	{attribute 'TcIecLibraryType'}
	{attribute 'external_name' := 'F_VN_Homography_GUID_BACE21C2_AF59_42BD_5B50_39109165FCFC'}
	(* Find the homography (perspective transformation) between two planar point sets. *)
	FUNCTION F_VN_Homography : HRESULT
	VAR_INPUT
		ipSrcPoints	:	ITcVnContainer;	(* Container with at least 4 source points (ContainerType_Vector_TcVnPoint2_REAL) *)
		ipDestPoints	:	ITcVnContainer;	(* Container with destination points (same number as ipSrcPoints, ContainerType_Vector_TcVnPoint2_REAL) *)
		aPerspectiveTransform	:	REFERENCE TO TcVnMatrix3x3_LREAL;	(* Returns the perspective transformation matrix, which transforms the source points to the destination points *)
		hrPrev	:	HRESULT;	(* HRESULT indicating the result of previous operations (If SUCCEEDED(hrPrev) equals false, no operation is executed.) *)
	END_VAR

END_FUNCTION

// Functions/Geometric and Coordinate Transformations/F_VN_HomographyExp

	{attribute 'TcIecLibraryType'}
	{attribute 'external_name' := 'F_VN_HomographyExp_GUID_957B3768_7821_437F_6422_7D349715F2AB'}
	(* Find the homography (perspective transformation) between two planar point sets. (expert function) *)
	FUNCTION F_VN_HomographyExp : HRESULT
	VAR_INPUT
		ipSrcPoints	:	ITcVnContainer;	(* Container with at least 4 source points (ContainerType_Vector_TcVnPoint2_REAL) *)
		ipDestPoints	:	ITcVnContainer;	(* Container with destination points (same number as ipSrcPoints, ContainerType_Vector_TcVnPoint2_REAL) *)
		aPerspectiveTransform	:	REFERENCE TO TcVnMatrix3x3_LREAL;	(* Returns the perspective transformation matrix, which transforms the source points to the destination points *)
		eAlgorithm	:	ETcVnEstimationAlgorithm;	(* Estimation algorithm *)
		fReprojThreshold	:	LREAL;	(* Maximum allowed reprojection error to treat a point pair as an inlier (only for RANSAC, RHO) *)
		ipInlierMask	:	REFERENCE TO ITcVnContainer;	(* Returns a mask marking the inliers (optional, set to 0 if not required; ContainerType_Vector_SINT; only for RANSAC, LMEDS) *)
		nMaxIterations	:	UDINT;	(* Maximum number of RANSAC iterations *)
		fConfidence	:	LREAL;	(* Confidence (0..1) *)
		hrPrev	:	HRESULT;	(* HRESULT indicating the result of previous operations (If SUCCEEDED(hrPrev) equals false, no operation is executed.) *)
	END_VAR

END_FUNCTION

// Functions/Geometric and Coordinate Transformations/F_VN_ImagePointsWorldDistance

	{attribute 'TcIecLibraryType'}
	{attribute 'external_name' := 'F_VN_ImagePointsWorldDistance_GUID_B7CC4CD8_D9B9_453D_47E9_DCE0997F3FF0'}
	(* Computes the distance in the world coordinate system between two points (in the same world coordinate z layer) given in image coordinates. *)
	FUNCTION F_VN_ImagePointsWorldDistance : HRESULT
	VAR_INPUT
		aImagePoint1	:	REFERENCE TO TcVnPoint2_REAL;	(* First point in the image coordinate system *)
		aImagePoint2	:	REFERENCE TO TcVnPoint2_REAL;	(* Second point in the image coordinate system *)
		fWorldDistance	:	REFERENCE TO LREAL;	(* Returns the distance between aImagePoint1 and aImagePoint2 in the world coordinate system *)
		aCameraMatrix	:	REFERENCE TO TcVnMatrix3x3_LREAL;	(* 3x3 camera matrix containing the intrinsic parameters *)
		aDistortionCoefficients	:	REFERENCE TO TcVnArray8_LREAL;	(* Lens distortion coefficients [k1, k2, p1, p2, k3, k4, k5, k6] *)
		aRotationMatrix	:	REFERENCE TO TcVnMatrix3x3_LREAL;	(* 3x3 rotation matrix *)
		aTranslationVector	:	REFERENCE TO TcVnVector3_LREAL;	(* Translation vector *)
		fZ	:	LREAL;	(* z coordinate (world coordinate system) of the given points (0 would be at (toplevel) calibration pattern) *)
		hrPrev	:	HRESULT;	(* HRESULT indicating the result of previous operations (If SUCCEEDED(hrPrev) equals false, no operation is executed.) *)
	END_VAR

END_FUNCTION

// Functions/Geometric and Coordinate Transformations/F_VN_InvertAffineTransformation

	{attribute 'TcIecLibraryType'}
	{attribute 'external_name' := 'F_VN_InvertAffineTransformation_GUID_9CD3C3CD_AED1_4AC7_6B76_3AB059F5DF24'}
	(* Invert a 2D affine transformation matrix. *)
	FUNCTION F_VN_InvertAffineTransformation : HRESULT
	VAR_INPUT
		aTransformationMatrix	:	REFERENCE TO TcVnMatrix2x3_LREAL;	(* Source affine transformation matrix *)
		aInvertedTransformationMatrix	:	REFERENCE TO TcVnMatrix2x3_LREAL;	(* Resulting inverted affine transformation matrix *)
		hrPrev	:	HRESULT;	(* HRESULT indicating the result of previous operations (If SUCCEEDED(hrPrev) equals false, no operation is executed.) *)
	END_VAR

END_FUNCTION

// Functions/Geometric and Coordinate Transformations/F_VN_PerspectiveTransformation

	{attribute 'TcIecLibraryType'}
	{attribute 'external_name' := 'F_VN_PerspectiveTransformation_GUID_A10BDBDF_3A4E_42F2_67E8_D12DFF09F118'}
	(* Apply a perspective transformation (rotation + translation, e.g. from extrinsic calibration) to 3D point coordinates. *)
	FUNCTION F_VN_PerspectiveTransformation : HRESULT
	VAR_INPUT
		ipSrcPoints	:	ITcVnContainer;	(* Container with 3D source points (TcVnPoint3_REAL or TcVnPoint3_LREAL) *)
		ipDestPoints	:	REFERENCE TO ITcVnContainer;	(* Returns the transformed points (same type as ipSrcPoints) *)
		aRotationMatrix	:	REFERENCE TO TcVnMatrix3x3_LREAL;	(* 3x3 rotation matrix *)
		aTranslationVector	:	REFERENCE TO TcVnVector3_LREAL;	(* Translation vector *)
		hrPrev	:	HRESULT;	(* HRESULT indicating the result of previous operations (If SUCCEEDED(hrPrev) equals false, no operation is executed.) *)
	END_VAR

END_FUNCTION

// Functions/Geometric and Coordinate Transformations/F_VN_PyramidDown

	{attribute 'TcIecLibraryType'}
	{attribute 'external_name' := 'F_VN_PyramidDown_GUID_A46C393D_F610_403D_7A8C_F077AAEC78D7'}
	(* Downsamples an image to half width and height. *)
	FUNCTION F_VN_PyramidDown : HRESULT
	VAR_INPUT
		ipSrcImage	:	ITcVnImage;	(* Source image *)
		ipDestImage	:	REFERENCE TO ITcVnImage;	(* Destination image (An appropriate destination image will be created if required.) *)
		hrPrev	:	HRESULT;	(* HRESULT indicating the result of previous operations (If SUCCEEDED(hrPrev) equals false, no operation is executed.) *)
	END_VAR

END_FUNCTION

// Functions/Geometric and Coordinate Transformations/F_VN_PyramidUp

	{attribute 'TcIecLibraryType'}
	{attribute 'external_name' := 'F_VN_PyramidUp_GUID_C7623CD4_6E7C_4659_6255_40F31BC5DBAD'}
	(* Upsamples an image to double width and height. *)
	FUNCTION F_VN_PyramidUp : HRESULT
	VAR_INPUT
		ipSrcImage	:	ITcVnImage;	(* Source image *)
		ipDestImage	:	REFERENCE TO ITcVnImage;	(* Destination image (An appropriate destination image will be created if required.) *)
		hrPrev	:	HRESULT;	(* HRESULT indicating the result of previous operations (If SUCCEEDED(hrPrev) equals false, no operation is executed.) *)
	END_VAR

END_FUNCTION

// Functions/Geometric and Coordinate Transformations/F_VN_RemapImageToLogPolarSpace

	{attribute 'TcIecLibraryType'}
	{attribute 'external_name' := 'F_VN_RemapImageToLogPolarSpace_GUID_317EBF55_4B2D_478D_5790_D67FEE90C80E'}
	(* Remap an image to log-polar space. *)
	FUNCTION F_VN_RemapImageToLogPolarSpace : HRESULT
	VAR_INPUT
		ipSrcImage	:	ITcVnImage;	(* Source image *)
		ipDestImage	:	REFERENCE TO ITcVnImage;	(* Destination image (Must not be the same as ipSrcImage! An appropriate destination image will be created if required.) *)
		aCenter	:	REFERENCE TO TcVnPoint2_REAL;	(* Center point for the transformation *)
		hrPrev	:	HRESULT;	(* HRESULT indicating the result of previous operations (If SUCCEEDED(hrPrev) equals false, no operation is executed.) *)
	END_VAR

END_FUNCTION

// Functions/Geometric and Coordinate Transformations/F_VN_RemapImageToLogPolarSpaceExp

	{attribute 'TcIecLibraryType'}
	{attribute 'external_name' := 'F_VN_RemapImageToLogPolarSpaceExp_GUID_C452CB02_0761_45C6_6145_95B8240BC99B'}
	(* Remap an image to log-polar space. (expert function) *)
	FUNCTION F_VN_RemapImageToLogPolarSpaceExp : HRESULT
	VAR_INPUT
		ipSrcImage	:	ITcVnImage;	(* Source image *)
		ipDestImage	:	REFERENCE TO ITcVnImage;	(* Destination image (Must not be the same as ipSrcImage! An appropriate destination image will be created if required.) *)
		aCenter	:	REFERENCE TO TcVnPoint2_REAL;	(* Center point for the transformation *)
		fScale	:	LREAL;	(* Magnitude scale parameter (set to 0 for auto select) *)
		eInterpolationType	:	ETcVnInterpolationType;	(* Interpolation type *)
		hrPrev	:	HRESULT;	(* HRESULT indicating the result of previous operations (If SUCCEEDED(hrPrev) equals false, no operation is executed.) *)
	END_VAR

END_FUNCTION

// Functions/Geometric and Coordinate Transformations/F_VN_RemapImageToPolarSpace

	{attribute 'TcIecLibraryType'}
	{attribute 'external_name' := 'F_VN_RemapImageToPolarSpace_GUID_81A2C6C8_42C0_4CD4_568D_C8E6F1DB1310'}
	(* Remap an image to polar space. *)
	FUNCTION F_VN_RemapImageToPolarSpace : HRESULT
	VAR_INPUT
		ipSrcImage	:	ITcVnImage;	(* Source image *)
		ipDestImage	:	REFERENCE TO ITcVnImage;	(* Destination image (Must not be the same as ipSrcImage! An appropriate destination image will be created if required.) *)
		aCenter	:	REFERENCE TO TcVnPoint2_REAL;	(* Center point for the transformation *)
		hrPrev	:	HRESULT;	(* HRESULT indicating the result of previous operations (If SUCCEEDED(hrPrev) equals false, no operation is executed.) *)
	END_VAR

END_FUNCTION

// Functions/Geometric and Coordinate Transformations/F_VN_RemapImageToPolarSpaceExp

	{attribute 'TcIecLibraryType'}
	{attribute 'external_name' := 'F_VN_RemapImageToPolarSpaceExp_GUID_C787DB85_1BF7_45E0_4B56_DABB0704543F'}
	(* Remap an image to polar space. (expert function) *)
	FUNCTION F_VN_RemapImageToPolarSpaceExp : HRESULT
	VAR_INPUT
		ipSrcImage	:	ITcVnImage;	(* Source image *)
		ipDestImage	:	REFERENCE TO ITcVnImage;	(* Destination image (Must not be the same as ipSrcImage! An appropriate destination image will be created if required.) *)
		aCenter	:	REFERENCE TO TcVnPoint2_REAL;	(* Center point for the transformation *)
		fMaxRadius	:	LREAL;	(* Maximum radius for the transformation (set to 0 for auto select) *)
		eInterpolationType	:	ETcVnInterpolationType;	(* Interpolation type *)
		hrPrev	:	HRESULT;	(* HRESULT indicating the result of previous operations (If SUCCEEDED(hrPrev) equals false, no operation is executed.) *)
	END_VAR

END_FUNCTION

// Functions/Geometric and Coordinate Transformations/F_VN_ResizeImage

	{attribute 'TcIecLibraryType'}
	{attribute 'external_name' := 'F_VN_ResizeImage_GUID_B297F5D8_147F_492A_69A8_8AF713B422F2'}
	(* Resize an image using a specific interpolation type. *)
	FUNCTION F_VN_ResizeImage : HRESULT
	VAR_INPUT
		ipSrcImage	:	ITcVnImage;	(* Source image *)
		ipDestImage	:	REFERENCE TO ITcVnImage;	(* Destination image (An appropriate image will be created if required.) *)
		nWidth	:	UDINT;	(* New width *)
		nHeight	:	UDINT;	(* New height *)
		eInterpolationType	:	ETcVnInterpolationType;	(* Interpolation type *)
		hrPrev	:	HRESULT;	(* HRESULT indicating the result of previous operations (If SUCCEEDED(hrPrev) equals false, no operation is executed.) *)
	END_VAR

END_FUNCTION

// Functions/Geometric and Coordinate Transformations/F_VN_RotateImage

	{attribute 'TcIecLibraryType'}
	{attribute 'external_name' := 'F_VN_RotateImage_GUID_D34C046F_1F65_490B_4694_D44E5095070F'}
	(* Rotate an image by 90, 180, or 270 degrees in clockwise direction. *)
	FUNCTION F_VN_RotateImage : HRESULT
	VAR_INPUT
		ipSrcImage	:	ITcVnImage;	(* Source image *)
		ipDestImage	:	REFERENCE TO ITcVnImage;	(* Destination image (An appropriate image will be created if required.) *)
		eAngle	:	ETcVnRotationAngle;	(* Rotation angle *)
		hrPrev	:	HRESULT;	(* HRESULT indicating the result of previous operations (If SUCCEEDED(hrPrev) equals false, no operation is executed.) *)
	END_VAR

END_FUNCTION

// Functions/Geometric and Coordinate Transformations/F_VN_WarpAffine

	{attribute 'TcIecLibraryType'}
	{attribute 'external_name' := 'F_VN_WarpAffine_GUID_2706E1B0_49AA_4EA6_4BCD_DBE188F95A14'}
	(* Apply an affine transformation to an image. *)
	FUNCTION F_VN_WarpAffine : HRESULT
	VAR_INPUT
		ipSrcImage	:	ITcVnImage;	(* Source image *)
		ipDestImage	:	REFERENCE TO ITcVnImage;	(* Destination image (An appropriate image will be created if required.) *)
		aTransformationMatrix	:	REFERENCE TO TcVnMatrix2x3_LREAL;	(* Affine transformation matrix *)
		hrPrev	:	HRESULT;	(* HRESULT indicating the result of previous operations (If SUCCEEDED(hrPrev) equals false, no operation is executed.) *)
	END_VAR

END_FUNCTION

// Functions/Geometric and Coordinate Transformations/F_VN_WarpAffineExp

	{attribute 'TcIecLibraryType'}
	{attribute 'external_name' := 'F_VN_WarpAffineExp_GUID_BA2CF855_8F8F_4276_5F6B_1E3D858121C1'}
	(* Apply an affine transformation to an image. (expert function) *)
	FUNCTION F_VN_WarpAffineExp : HRESULT
	VAR_INPUT
		ipSrcImage	:	ITcVnImage;	(* Source image *)
		ipDestImage	:	REFERENCE TO ITcVnImage;	(* Destination image (An appropriate image will be created if required.) *)
		aTransformationMatrix	:	REFERENCE TO TcVnMatrix2x3_LREAL;	(* Affine transformation matrix *)
		nDestWidth	:	UDINT;	(* Width of the destination image *)
		nDestHeight	:	UDINT;	(* Height of the destination image *)
		eInterpolationType	:	ETcVnInterpolationType;	(* Interpolation method *)
		bWarpInverse	:	BOOL;	(* Handle aTransformationMatrix as the inverse transformation *)
		eBorderInterpolation	:	ETcVnBorderInterpolationMethod;	(* Border interpolation method (ISOLATED not supported) *)
		fBorderValue	:	LREAL;	(* Border value, if CONSTANT is used *)
		hrPrev	:	HRESULT;	(* HRESULT indicating the result of previous operations (If SUCCEEDED(hrPrev) equals false, no operation is executed.) *)
	END_VAR

END_FUNCTION

// Functions/Geometric and Coordinate Transformations/F_VN_WarpAffine_Container

	{attribute 'TcIecLibraryType'}
	{attribute 'external_name' := 'F_VN_WarpAffine_Container_GUID_E245EF6B_F4F8_40CB_6A97_91315828A7CE'}
	(* Apply an affine transformation to a container of 2D points. *)
	FUNCTION F_VN_WarpAffine_Container : HRESULT
	VAR_INPUT
		ipSrcPoints	:	ITcVnContainer;	(* Source points (ContainerType_Vector_TcVnPoint2_DINT or ContainerType_Vector_TcVnPoint2_REAL or ContainerType_Vector_TcVnPoint2_LREAL) *)
		ipDestPoints	:	REFERENCE TO ITcVnContainer;	(* Returns the transformed points (same type ID as ipSrcPoints; Non-zero interface pointers are reused.) *)
		aTransformationMatrix	:	REFERENCE TO TcVnMatrix2x3_LREAL;	(* Affine transformation matrix *)
		hrPrev	:	HRESULT;	(* HRESULT indicating the result of previous operations (If SUCCEEDED(hrPrev) equals false, no operation is executed.) *)
	END_VAR

END_FUNCTION

// Functions/Geometric and Coordinate Transformations/F_VN_WarpAffine_Point

	{attribute 'TcIecLibraryType'}
	{attribute 'external_name' := 'F_VN_WarpAffine_Point_GUID_5382904B_C8E3_45B3_56E2_503ADF42779C'}
	(* Apply an affine transformation to a 2D point. *)
	FUNCTION F_VN_WarpAffine_Point : HRESULT
	VAR_INPUT
		aSrcPoint	:	REFERENCE TO TcVnPoint2_LREAL;	(* Source point *)
		aDestPoint	:	REFERENCE TO TcVnPoint2_LREAL;	(* Destination point *)
		aTransformationMatrix	:	REFERENCE TO TcVnMatrix2x3_LREAL;	(* Affine transformation matrix *)
		hrPrev	:	HRESULT;	(* HRESULT indicating the result of previous operations (If SUCCEEDED(hrPrev) equals false, no operation is executed.) *)
	END_VAR

END_FUNCTION

// Functions/Geometric and Coordinate Transformations/F_VN_WarpPerspective

	{attribute 'TcIecLibraryType'}
	{attribute 'external_name' := 'F_VN_WarpPerspective_GUID_A5B0ACEA_FF20_43BC_4699_A7DC79225D3D'}
	(* Apply a perspective transformation to an image. *)
	FUNCTION F_VN_WarpPerspective : HRESULT
	VAR_INPUT
		ipSrcImage	:	ITcVnImage;	(* Source image *)
		ipDestImage	:	REFERENCE TO ITcVnImage;	(* Destination image (An appropriate image will be created if required.) *)
		aTransformationMatrix	:	REFERENCE TO TcVnMatrix3x3_LREAL;	(* Perspective transformation matrix *)
		hrPrev	:	HRESULT;	(* HRESULT indicating the result of previous operations (If SUCCEEDED(hrPrev) equals false, no operation is executed.) *)
	END_VAR

END_FUNCTION

// Functions/Geometric and Coordinate Transformations/F_VN_WarpPerspectiveExp

	{attribute 'TcIecLibraryType'}
	{attribute 'external_name' := 'F_VN_WarpPerspectiveExp_GUID_5EE68E40_2F06_46A9_53D0_6833136D40D3'}
	(* Apply a perspective transformation to an image. (expert function) *)
	FUNCTION F_VN_WarpPerspectiveExp : HRESULT
	VAR_INPUT
		ipSrcImage	:	ITcVnImage;	(* Source image *)
		ipDestImage	:	REFERENCE TO ITcVnImage;	(* Destination image (An appropriate image will be created if required.) *)
		aTransformationMatrix	:	REFERENCE TO TcVnMatrix3x3_LREAL;	(* Perspective transformation matrix *)
		nDestWidth	:	UDINT;	(* Width of the destination image *)
		nDestHeight	:	UDINT;	(* Height of the destination image *)
		eInterpolationType	:	ETcVnInterpolationType;	(* Interpolation method *)
		bWarpInverse	:	BOOL;	(* Handle aTransformationMatrix as the inverse transformation *)
		eBorderInterpolation	:	ETcVnBorderInterpolationMethod;	(* Border interpolation method (ISOLATED not supported) *)
		fBorderValue	:	LREAL;	(* Border value, if CONSTANT is used *)
		hrPrev	:	HRESULT;	(* HRESULT indicating the result of previous operations (If SUCCEEDED(hrPrev) equals false, no operation is executed.) *)
	END_VAR

END_FUNCTION

// Functions/Geometric and Coordinate Transformations/F_VN_WarpPerspective_Point

	{attribute 'TcIecLibraryType'}
	{attribute 'external_name' := 'F_VN_WarpPerspective_Point_GUID_5538B106_075B_440A_4CE3_92BE11A2EC15'}
	(* Apply a perspective transformation to a 2D point. *)
	FUNCTION F_VN_WarpPerspective_Point : HRESULT
	VAR_INPUT
		aSrcPoint	:	REFERENCE TO TcVnPoint2_LREAL;	(* Source point *)
		aDestPoint	:	REFERENCE TO TcVnPoint2_LREAL;	(* Destination point *)
		aTransformationMatrix	:	REFERENCE TO TcVnMatrix3x3_LREAL;	(* Perspective transformation matrix *)
		hrPrev	:	HRESULT;	(* HRESULT indicating the result of previous operations (If SUCCEEDED(hrPrev) equals false, no operation is executed.) *)
	END_VAR

END_FUNCTION

// Functions/Contour Analysis/F_VN_ApproximatePolygon

	{attribute 'TcIecLibraryType'}
	{attribute 'external_name' := 'F_VN_ApproximatePolygon_GUID_CC2021C4_5F20_4D4F_750B_DA13A9B816C9'}
	(* Approximate a contour to a simplified polygon (using the Douglas-Peucker algorithm). *)
	FUNCTION F_VN_ApproximatePolygon : HRESULT
	VAR_INPUT
		ipSrcContour	:	ITcVnContainer;	(* Single contour (ContainerType_Vector_TcVnPoint2_DINT or ContainerType_Vector_TcVnPoint2_REAL; The elements of this container are the points of the contour.) *)
		ipDestContour	:	REFERENCE TO ITcVnContainer;	(* Returns a container which is filled with the approximated polygon points (same type ID as ipSrcContour; Non-zero interface pointers are reused.) *)
		fMaxDist	:	LREAL;	(* Maximum distance between the original contour and its approximation *)
		bClosed	:	BOOL;	(* Specify, if the contour is closed (first and last points connected) or not *)
		hrPrev	:	HRESULT;	(* HRESULT indicating the result of previous operations (If SUCCEEDED(hrPrev) equals false, no operation is executed.) *)
	END_VAR

END_FUNCTION

// Functions/Contour Analysis/F_VN_CheckIfPointIsInsideContour

	{attribute 'TcIecLibraryType'}
	{attribute 'external_name' := 'F_VN_CheckIfPointIsInsideContour_GUID_0925219F_5855_4324_6916_36F829EC1C7B'}
	(* Checks if a point is inside a contour (and optionally return the distance to it). *)
	FUNCTION F_VN_CheckIfPointIsInsideContour : HRESULT
	VAR_INPUT
		ipContour	:	ITcVnContainer;	(* Single contour (ContainerType_Vector_TcVnPoint2_DINT or ContainerType_Vector_TcVnPoint2_REAL) *)
		aPoint	:	REFERENCE TO TcVnPoint2_REAL;	(* Point position to check *)
		fDist	:	REFERENCE TO LREAL;	(* Returns the result (> 0: the point is inside the contour; 0: the point is on the contour; < 0: the point is outside the contour) *)
		bMeasureDistance	:	BOOL;	(* If true, fDist returns the distance to the nearest contour edge. Otherwise, fDist only returns -1, 0 or +1 (recommended to set to false if the distance is not required, as this is faster). *)
		hrPrev	:	HRESULT;	(* HRESULT indicating the result of previous operations (If SUCCEEDED(hrPrev) equals false, no operation is executed.) *)
	END_VAR

END_FUNCTION

// Functions/Contour Analysis/F_VN_ContourArea

	{attribute 'TcIecLibraryType'}
	{attribute 'external_name' := 'F_VN_ContourArea_GUID_D8EF7B56_DDD8_4A2A_43D3_6C64F8AEA3E5'}
	(* Estimate the contour area using Green's formula. *)
	FUNCTION F_VN_ContourArea : HRESULT
	VAR_INPUT
		ipContour	:	ITcVnContainer;	(* Single contour (ContainerType_Vector_TcVnPoint2_DINT or ContainerType_Vector_TcVnPoint2_REAL; The elements of this container are the points of the contour.) *)
		fArea	:	REFERENCE TO LREAL;	(* Returns the estimated contour area (The actual contour area may differ depending on the shape of the contour.) *)
		hrPrev	:	HRESULT;	(* HRESULT indicating the result of previous operations (If SUCCEEDED(hrPrev) equals false, no operation is executed.) *)
	END_VAR

END_FUNCTION

// Functions/Contour Analysis/F_VN_ContourCenterOfMass

	{attribute 'TcIecLibraryType'}
	{attribute 'external_name' := 'F_VN_ContourCenterOfMass_GUID_648B2107_798D_4ED5_549A_9A87656EE4D8'}
	(* Computes the center of mass of a contour. *)
	FUNCTION F_VN_ContourCenterOfMass : HRESULT
	VAR_INPUT
		ipContour	:	ITcVnContainer;	(* Single contour (ContainerType_Vector_TcVnPoint2_DINT or ContainerType_Vector_TcVnPoint2_REAL; The elements of this container are the points of the contour.) *)
		aCenterOfMass	:	REFERENCE TO TcVnPoint2_LREAL;	(* Returns the center of mass of the contour *)
		hrPrev	:	HRESULT;	(* HRESULT indicating the result of previous operations (If SUCCEEDED(hrPrev) equals false, no operation is executed.) *)
	END_VAR

END_FUNCTION

// Functions/Contour Analysis/F_VN_ContourCircularity

	{attribute 'TcIecLibraryType'}
	{attribute 'external_name' := 'F_VN_ContourCircularity_GUID_9E609700_7C0A_461F_5A42_99C7290586FE'}
	(* Computes the circularity of a contour (1.0: ideal circle, 0.0: straight line). *)
	FUNCTION F_VN_ContourCircularity : HRESULT
	VAR_INPUT
		ipContour	:	ITcVnContainer;	(* Single contour (ContainerType_Vector_TcVnPoint2_DINT or ContainerType_Vector_TcVnPoint2_REAL; The elements of this container are the points of the contour.) *)
		fCircularity	:	REFERENCE TO LREAL;	(* Returns the circularity of the contour [0..1] *)
		hrPrev	:	HRESULT;	(* HRESULT indicating the result of previous operations (If SUCCEEDED(hrPrev) equals false, no operation is executed.) *)
	END_VAR

END_FUNCTION

// Functions/Contour Analysis/F_VN_ContourEccentricity

	{attribute 'TcIecLibraryType'}
	{attribute 'external_name' := 'F_VN_ContourEccentricity_GUID_FFD20AEF_8984_4F5E_766E_3023FBFF4334'}
	(* Computes the eccentricity of a contour (0.0: circular, 1.0: linear). *)
	FUNCTION F_VN_ContourEccentricity : HRESULT
	VAR_INPUT
		ipContour	:	ITcVnContainer;	(* Single contour (ContainerType_Vector_TcVnPoint2_DINT or ContainerType_Vector_TcVnPoint2_REAL; The elements of this container are the points of the contour.) *)
		fEccentricity	:	REFERENCE TO LREAL;	(* Returns the eccentricity of the contour [0..1] *)
		hrPrev	:	HRESULT;	(* HRESULT indicating the result of previous operations (If SUCCEEDED(hrPrev) equals false, no operation is executed.) *)
	END_VAR

END_FUNCTION

// Functions/Contour Analysis/F_VN_ContourExtremePoint

	{attribute 'TcIecLibraryType'}
	{attribute 'external_name' := 'F_VN_ContourExtremePoint_GUID_8F761823_6FFC_4019_7B5F_2B40F751511F'}
	(* Finds the contour extreme point. *)
	FUNCTION F_VN_ContourExtremePoint : HRESULT
	VAR_INPUT
		ipContour	:	ITcVnContainer;	(* Source container with 2D points (TcVnPoint2_DINT or TcVnPoint2_REAL or TcVnPoint2_LREAL) *)
		eDirection	:	ETcVnExtremePointDirection;	(* Selects the search direction for the extreme point *)
		aExtremePoint	:	REFERENCE TO TcVnPoint2_LREAL;	(* Returns the extreme point of the contour, according to eDirection *)
		hrPrev	:	HRESULT;	(* HRESULT indicating the result of previous operations (If SUCCEEDED(hrPrev) equals false, no operation is executed.) *)
	END_VAR

END_FUNCTION

// Functions/Contour Analysis/F_VN_ContourMoments

	{attribute 'TcIecLibraryType'}
	{attribute 'external_name' := 'F_VN_ContourMoments_GUID_FAC9EEF4_5569_47FA_777B_374334F5BD38'}
	(* Computes the spatial moments, the central moments, and the central normalized moments of a contour up to the third order. *)
	FUNCTION F_VN_ContourMoments : HRESULT
	VAR_INPUT
		ipContour	:	ITcVnContainer;	(* Single contour (ContainerType_Vector_TcVnPoint2_DINT or ContainerType_Vector_TcVnPoint2_REAL; The elements of this container are the points of the contour.) *)
		stMoments	:	REFERENCE TO TcVnMoments;	(* Returns a struct containing the moments *)
		hrPrev	:	HRESULT;	(* HRESULT indicating the result of previous operations (If SUCCEEDED(hrPrev) equals false, no operation is executed.) *)
	END_VAR

END_FUNCTION

// Functions/Contour Analysis/F_VN_ContourPerimeter

	{attribute 'TcIecLibraryType'}
	{attribute 'external_name' := 'F_VN_ContourPerimeter_GUID_CA52E6A1_DDEA_4337_739C_F63A5F171A5F'}
	(* Computes the perimeter of a contour (curve length if the contour is not closed). *)
	FUNCTION F_VN_ContourPerimeter : HRESULT
	VAR_INPUT
		ipContour	:	ITcVnContainer;	(* Single contour (ContainerType_Vector_TcVnPoint2_DINT or ContainerType_Vector_TcVnPoint2_REAL; The elements of this container are the points of the contour.) *)
		fPerimeter	:	REFERENCE TO LREAL;	(* Returns the perimeter of the contour *)
		bClosed	:	BOOL;	(* Specifys, if the contour is closed (first and last points connected) or not *)
		hrPrev	:	HRESULT;	(* HRESULT indicating the result of previous operations (If SUCCEEDED(hrPrev) equals false, no operation is executed.) *)
	END_VAR

END_FUNCTION

// Functions/Contour Analysis/F_VN_ContourRoundness

	{attribute 'TcIecLibraryType'}
	{attribute 'external_name' := 'F_VN_ContourRoundness_GUID_0921D745_4FBD_4A8F_6DB5_7FBDA3359228'}
	(* Computes the roundness of a contour (perimeter^2 / area). *)
	FUNCTION F_VN_ContourRoundness : HRESULT
	VAR_INPUT
		ipContour	:	ITcVnContainer;	(* Single contour (ContainerType_Vector_TcVnPoint2_DINT or ContainerType_Vector_TcVnPoint2_REAL; The elements of this container are the points of the contour.) *)
		fRoundness	:	REFERENCE TO LREAL;	(* Returns the roundness of the contour *)
		hrPrev	:	HRESULT;	(* HRESULT indicating the result of previous operations (If SUCCEEDED(hrPrev) equals false, no operation is executed.) *)
	END_VAR

END_FUNCTION

// Functions/Contour Analysis/F_VN_ConvexHullPoints

	{attribute 'TcIecLibraryType'}
	{attribute 'external_name' := 'F_VN_ConvexHullPoints_GUID_5386C16C_F8EA_4A71_7709_FBD086BD9B3C'}
	(* Determines the convex hull of a point set. *)
	FUNCTION F_VN_ConvexHullPoints : HRESULT
	VAR_INPUT
		ipPointSet	:	ITcVnContainer;	(* Source point set (ContainerType_Vector_TcVnPoint2_DINT or ContainerType_Vector_TcVnPoint2_REAL; The elements of this container are the individual points.) *)
		ipConvexHull	:	REFERENCE TO ITcVnContainer;	(* Returns a container which is filled with the sorted convex hull points (same type ID as ipPointSet; Non-zero interface pointers are reused.) *)
		hrPrev	:	HRESULT;	(* HRESULT indicating the result of previous operations (If SUCCEEDED(hrPrev) equals false, no operation is executed.) *)
	END_VAR

END_FUNCTION

// Functions/Contour Analysis/F_VN_ConvexHullPointsExp

	{attribute 'TcIecLibraryType'}
	{attribute 'external_name' := 'F_VN_ConvexHullPointsExp_GUID_1E36CE0E_A49C_4D24_4893_7EDE50EB52D5'}
	(* Determines the convex hull of a point set. (expert function) *)
	FUNCTION F_VN_ConvexHullPointsExp : HRESULT
	VAR_INPUT
		ipPointSet	:	ITcVnContainer;	(* Source point set (ContainerType_Vector_TcVnPoint2_DINT or ContainerType_Vector_TcVnPoint2_REAL; The elements of this container are the individual points.) *)
		ipConvexHull	:	REFERENCE TO ITcVnContainer;	(* Returns a container which is filled with the sorted convex hull points (same type ID as ipPointSet; Non-zero interface pointers are reused.) *)
		bClockwise	:	BOOL;	(* Selects the sorting direction of the hull points, assuming cartesian coordinates. *)
		hrPrev	:	HRESULT;	(* HRESULT indicating the result of previous operations (If SUCCEEDED(hrPrev) equals false, no operation is executed.) *)
	END_VAR

END_FUNCTION

// Functions/Contour Analysis/F_VN_CustomElementWiseContainerOperation_ITcVnContainer

	{attribute 'TcIecLibraryType'}
	{attribute 'external_name' := 'F_VN_CustomElementWiseContainerOperation_ITcVnContainer_GUID_8B5FFCB6_72C1_4217_42F9_2485E219D315'}
	(* Performs a custom, element wise operation on a set of up to 3 containers. *)
	FUNCTION F_VN_CustomElementWiseContainerOperation_ITcVnContainer : HRESULT
	VAR_INPUT
		ipContainer1	:	ITcVnContainer;	(* Container 1 *)
		ipContainer2	:	ITcVnContainer;	(* Container 2 *)
		ipContainer3	:	ITcVnContainer;	(* Container 3 *)
		ipOperationFB	:	ITcVnCustomContainerOperation_ITcVnContainer;	(* Custom operation on the container elements *)
		hrPrev	:	HRESULT;	(* HRESULT indicating the result of previous operations (If SUCCEEDED(hrPrev) equals false, no operation is executed.) *)
	END_VAR

END_FUNCTION

// Interfaces/Containers/Function Blocks/ITcVnCustomContainerOperation_ITcVnContainer

	(* Offers an interface for custom, elementwise container operations (for containers of containers) with up to 3 different containers. *)
	{attribute 'c++_compatible'}
	INTERFACE ITcVnCustomContainerOperation_ITcVnContainer


(* Executes the custom operation on the container elements. *)
	{attribute 'c++_compatible'}
	{attribute 'minimal_input_size' := '4'}
	{attribute 'pack_mode' := '4'}
	METHOD Execute : HRESULT
	VAR_INPUT
		ipElement1 : ITcVnContainer;
		ipElement2 : ITcVnContainer;
		ipElement3 : ITcVnContainer;
	END_VAR
END_METHOD

END_INTERFACE

// Functions/Contour Analysis/F_VN_CustomElementWiseContainerOperation_ITcVnForwardIterator

	{attribute 'TcIecLibraryType'}
	{attribute 'external_name' := 'F_VN_CustomElementWiseContainerOperation_ITcVnForwardIterator_GUID_A3F5CA41_1335_4213_550C_04C31E4F67AC'}
	(* Performs a custom, element wise operation on a set of up to 3 containers. *)
	FUNCTION F_VN_CustomElementWiseContainerOperation_ITcVnForwardIterator : HRESULT
	VAR_INPUT
		ipContainer1	:	ITcVnContainer;	(* Container 1 *)
		ipContainer2	:	ITcVnContainer;	(* Container 2 *)
		ipContainer3	:	ITcVnContainer;	(* Container 3 *)
		ipOperationFB	:	ITcVnCustomContainerOperation_ITcVnForwardIterator;	(* Custom operation on the elements *)
		hrPrev	:	HRESULT;	(* HRESULT indicating the result of previous operations (If SUCCEEDED(hrPrev) equals false, no operation is executed.) *)
	END_VAR

END_FUNCTION

// Interfaces/Containers/Function Blocks/ITcVnCustomContainerOperation_ITcVnForwardIterator

	(* Offers an interface for custom, elementwise container operations with up to 3 different containers. *)
	{attribute 'c++_compatible'}
	INTERFACE ITcVnCustomContainerOperation_ITcVnForwardIterator


(* Executes the custom operation on the container elements. *)
	{attribute 'c++_compatible'}
	{attribute 'minimal_input_size' := '4'}
	{attribute 'pack_mode' := '4'}
	METHOD Execute : HRESULT
	VAR_INPUT
		ipElement1 : ITcVnForwardIterator;
		ipElement2 : ITcVnForwardIterator;
		ipElement3 : ITcVnForwardIterator;
	END_VAR
END_METHOD

END_INTERFACE

// Functions/Contour Analysis/F_VN_EnclosingCircle

	{attribute 'TcIecLibraryType'}
	{attribute 'external_name' := 'F_VN_EnclosingCircle_GUID_2C49C5FC_5376_4B84_430E_36F041A3B079'}
	(* Searchs for a minimum area circle enclosing a set of points. *)
	FUNCTION F_VN_EnclosingCircle : HRESULT
	VAR_INPUT
		ipPointSet	:	ITcVnContainer;	(* Source point set (ContainerType_Vector_TcVnPoint2_DINT or ContainerType_Vector_TcVnPoint2_REAL; The elements of this container are the individual points.) *)
		aCenter	:	REFERENCE TO TcVnPoint2_REAL;	(* Returns the center of the circle *)
		fRadius	:	REFERENCE TO REAL;	(* Returns the radius of the circle *)
		hrPrev	:	HRESULT;	(* HRESULT indicating the result of previous operations (If SUCCEEDED(hrPrev) equals false, no operation is executed.) *)
	END_VAR

END_FUNCTION

// Functions/Contour Analysis/F_VN_EnclosingRectangle

	{attribute 'TcIecLibraryType'}
	{attribute 'external_name' := 'F_VN_EnclosingRectangle_GUID_5A1EA58F_F461_4FEB_5B48_1702EB63B7F9'}
	(* Searches for a minimum area rectangle enclosing a set of points. *)
	FUNCTION F_VN_EnclosingRectangle : HRESULT
	VAR_INPUT
		ipPointSet	:	ITcVnContainer;	(* Source point set (ContainerType_Vector_TcVnPoint2_DINT or ContainerType_Vector_TcVnPoint2_REAL; The elements of this container are the individual points.) *)
		stRectangle	:	REFERENCE TO TcVnRotatedRectangle;	(* Returns the determined rectangle *)
		hrPrev	:	HRESULT;	(* HRESULT indicating the result of previous operations (If SUCCEEDED(hrPrev) equals false, no operation is executed.) *)
	END_VAR

END_FUNCTION

// Functions/Contour Analysis/F_VN_EnclosingTriangle

	{attribute 'TcIecLibraryType'}
	{attribute 'external_name' := 'F_VN_EnclosingTriangle_GUID_97E20FD1_288B_4194_7EE7_758B19CB2E03'}
	(* Searches for a minimum area triangle enclosing a set of points. *)
	FUNCTION F_VN_EnclosingTriangle : HRESULT
	VAR_INPUT
		ipPointSet	:	ITcVnContainer;	(* Source point set (ContainerType_Vector_TcVnPoint2_DINT or ContainerType_Vector_TcVnPoint2_REAL; The elements of this container are the individual points.) *)
		aTriangleVertices	:	REFERENCE TO TcVnArray3_Point2_REAL;	(* Returns the 3 triangle vertices *)
		hrPrev	:	HRESULT;	(* HRESULT indicating the result of previous operations (If SUCCEEDED(hrPrev) equals false, no operation is executed.) *)
	END_VAR
	VAR_OUTPUT
		fArea	:	LREAL;	(* Returns the triangle area *)
	END_VAR

END_FUNCTION

// Functions/Contour Analysis/F_VN_FitEllipse

	{attribute 'TcIecLibraryType'}
	{attribute 'external_name' := 'F_VN_FitEllipse_GUID_9156269E_A5A1_4B36_427A_9C0D7756DE4D'}
	(* Fit an ellipse in a point set. *)
	FUNCTION F_VN_FitEllipse : HRESULT
	VAR_INPUT
		ipPointSet	:	ITcVnContainer;	(* Source point set (ContainerType_Vector_TcVnPoint2_DINT or ContainerType_Vector_TcVnPoint2_REAL; At least 5 reasonable points are required! The elements of this container are the individual points.) *)
		stEllipse	:	REFERENCE TO TcVnRotatedRectangle;	(* Resulting ellipse, described by a rotated rectangle. *)
		hrPrev	:	HRESULT;	(* HRESULT indicating the result of previous operations (If SUCCEEDED(hrPrev) equals false, no operation is executed.) *)
	END_VAR

END_FUNCTION

// Functions/Contour Analysis/F_VN_FitLine

	{attribute 'TcIecLibraryType'}
	{attribute 'external_name' := 'F_VN_FitLine_GUID_B14090CF_9687_4001_679C_C759C5707FE8'}
	(* Fit a line into a point set. *)
	FUNCTION F_VN_FitLine : HRESULT
	VAR_INPUT
		ipPointSet	:	ITcVnContainer;	(* Source point set (ContainerType_Vector_TcVnPoint2_DINT or ContainerType_Vector_TcVnPoint2_REAL; The elements of this container are the individual points.) *)
		aFitLine	:	REFERENCE TO TcVnVector4_LREAL;	(* Resulting line. The first and second element describe the x and y component of a vector collinear to the line. The third and fourth element describe the x and y component of a point on the line. *)
		hrPrev	:	HRESULT;	(* HRESULT indicating the result of previous operations (If SUCCEEDED(hrPrev) equals false, no operation is executed.) *)
	END_VAR

END_FUNCTION

// Functions/Contour Analysis/F_VN_FitLineExp

	{attribute 'TcIecLibraryType'}
	{attribute 'external_name' := 'F_VN_FitLineExp_GUID_798B9535_B3AC_4BA6_5F20_094D109DC99C'}
	(* Fit a line into a point set. (expert function) *)
	FUNCTION F_VN_FitLineExp : HRESULT
	VAR_INPUT
		ipPointSet	:	ITcVnContainer;	(* Source point set (ContainerType_Vector_TcVnPoint2_DINT or ContainerType_Vector_TcVnPoint2_REAL; The elements of this container are the individual points.) *)
		aFitLine	:	REFERENCE TO TcVnVector4_LREAL;	(* Resulting line. The first and second element describe the x and y component of a vector collinear to the line. The third and fourth element describe the x and y component of a point on the line. *)
		eDistanceType	:	ETcVnDistanceType;	(* Distance computation method (supported: L1, L2, L12, FAIR, WELSCH, HUBER) *)
		fParam	:	LREAL;	(* Numerical parameter (c) for some eDistanceType (should be >= 0). If 0, an optimal value is chosen internally. *)
		fEpsRadius	:	LREAL;	(* Accuracy of the radius (distance of the line from the coordinate origin, should be > 0). A smaller value means higher accuracy. *)
		fEpsAngle	:	LREAL;	(* Accuracy of the angle (should be > 0). A smaller value means higher accuracy. *)
		hrPrev	:	HRESULT;	(* HRESULT indicating the result of previous operations (If SUCCEEDED(hrPrev) equals false, no operation is executed.) *)
	END_VAR

END_FUNCTION

// Functions/Contour Analysis/F_VN_MatchContours

	{attribute 'TcIecLibraryType'}
	{attribute 'external_name' := 'F_VN_MatchContours_GUID_C7BA4036_D390_476A_71D5_3E2FD7EB1DC5'}
	(* Compare contours using the Hu moment invariants. In case of multiple contours in each container, the best matches are found and the average dissimilarity over all matched contours is returned. *)
	FUNCTION F_VN_MatchContours : HRESULT
	VAR_INPUT
		ipContour1	:	ITcVnContainer;	(* First contour (ContainerType_Vector_TcVnPoint2_DINT or ContainerType_Vector_TcVnPoint2_REAL; The elements of this container are the points of the contour) or collection of multiple contours (ContainerType_Vector_Vector_TcVnPoint2_DINT) *)
		ipContour2	:	ITcVnContainer;	(* Second contour (same type as ipContour1) *)
		eComparisonMethod	:	ETcVnContoursMatchComparisonMethod;	(* Method used for comparing the Hu moment invariants of the contours *)
		fDissimilarity	:	REFERENCE TO LREAL;	(* Returns the dissimilarity of the contours depending on the chosen comparison method *)
		hrPrev	:	HRESULT;	(* HRESULT indicating the result of previous operations (If SUCCEEDED(hrPrev) equals false, no operation is executed.) *)
	END_VAR

END_FUNCTION

// Functions/Contour Analysis/F_VN_MatchContoursExp

	{attribute 'TcIecLibraryType'}
	{attribute 'external_name' := 'F_VN_MatchContoursExp_GUID_B6C17942_DC1C_4F72_7734_5ABAF567D5A2'}
	(* Compare contours using the Hu moment invariants (and optionally further aspects). In case of multiple contours in each container, the best matches are found and the average dissimilarity over all matched contours is returned. (expert function) *)
	FUNCTION F_VN_MatchContoursExp : HRESULT
	VAR_INPUT
		ipContour1	:	ITcVnContainer;	(* First contour (ContainerType_Vector_TcVnPoint2_DINT or ContainerType_Vector_TcVnPoint2_REAL; The elements of this container are the points of the contour) or collection of multiple contours (ContainerType_Vector_Vector_TcVnPoint2_DINT) *)
		ipContour2	:	ITcVnContainer;	(* Second contour (same type as ipContour1) *)
		eComparisonMethod	:	ETcVnContoursMatchComparisonMethod;	(* Method used for comparing the Hu moment invariants of the contours *)
		fDissimilarity	:	REFERENCE TO LREAL;	(* Returns the dissimilarity of the contours depending on the chosen comparison method *)
		fAreaFactor	:	LREAL;	(* If > 0, the relative area difference between contours is scaled by this factor and added to the computed dissimilarity *)
		fAbsPositionFactor	:	LREAL;	(* If > 0, the absolute position difference between contours (i.e. the coordinates of the geometric contour centers) is scaled by this factor and added to the computed dissimilarity *)
		fRelPositionFactor	:	LREAL;	(* If > 0, the relative position difference between contours is scaled by this factor and added to the computed dissimilarity (only used if matching multiple contours) *)
		fNumDiffFactor	:	LREAL;	(* If > 0, the difference between the number of contours in both containers is scaled by this factor and added to the computed dissimilarity (only used if matching multiple contours) *)
		hrPrev	:	HRESULT;	(* HRESULT indicating the result of previous operations (If SUCCEEDED(hrPrev) equals false, no operation is executed.) *)
	END_VAR

END_FUNCTION

// Functions/Contour Analysis/F_VN_MatchContours1vsN

	{attribute 'TcIecLibraryType'}
	{attribute 'external_name' := 'F_VN_MatchContours1vsN_GUID_7E8CEC29_A31F_4D40_460D_DD6ACC817CE0'}
	(* Compare a reference contour with multiple other contours using the Hu moment invariants. Returns a sorted list of best matches. *)
	FUNCTION F_VN_MatchContours1vsN : HRESULT
	VAR_INPUT
		ipRefContour	:	ITcVnContainer;	(* Reference contour (ContainerType_Vector_TcVnPoint2_DINT or ContainerType_Vector_TcVnPoint2_REAL; The elements of this container are the points of the contour) *)
		ipContours	:	ITcVnContainer;	(* Collection of multiple contours (CTcVnContainer_Vector_Vector_TcVnPoint2_DINT) *)
		ipMatchIndexes	:	REFERENCE TO ITcVnContainer;	(* Returns the indexes of the best matches (CTcVnContainer_Vector_ULINT; sorted, first element is best match, i.e. has lowest dissimilarity) *)
		ipDissimilarities	:	REFERENCE TO ITcVnContainer;	(* Returns the computed dissimilarities of the best matches (CTcVnContainer_Vector_LREAL; Optional, set to 0 if not required; sorted corresponding to ipMatchIndexes) *)
		fDissimilarityThreshold	:	LREAL;	(* Neglect irrelevant matches, i.e. dissimilarity > fDissimilarityThreshold *)
		eComparisonMethod	:	ETcVnContoursMatchComparisonMethod;	(* Method used for comparing the Hu moment invariants of the contours *)
		hrPrev	:	HRESULT;	(* HRESULT indicating the result of previous operations (If SUCCEEDED(hrPrev) equals false, no operation is executed.) *)
	END_VAR

END_FUNCTION

// Functions/Contour Analysis/F_VN_MatchContours1vsNExp

	{attribute 'TcIecLibraryType'}
	{attribute 'external_name' := 'F_VN_MatchContours1vsNExp_GUID_33D890CC_2D47_4649_760A_F970590E77AD'}
	(* Compare a reference contour with multiple other contours using the Hu moment invariants (and optionally further aspects). Returns a sorted list of best matches. (expert function) *)
	FUNCTION F_VN_MatchContours1vsNExp : HRESULT
	VAR_INPUT
		ipRefContour	:	ITcVnContainer;	(* Reference contour (ContainerType_Vector_TcVnPoint2_DINT or ContainerType_Vector_TcVnPoint2_REAL; The elements of this container are the points of the contour) *)
		ipContours	:	ITcVnContainer;	(* Collection of multiple contours (CTcVnContainer_Vector_Vector_TcVnPoint2_DINT) *)
		ipMatchIndexes	:	REFERENCE TO ITcVnContainer;	(* Returns the indexes of the best matches (CTcVnContainer_Vector_ULINT; sorted, first element is best match, i.e. has lowest dissimilarity) *)
		ipDissimilarities	:	REFERENCE TO ITcVnContainer;	(* Returns the computed dissimilarities of the best matches (CTcVnContainer_Vector_LREAL; Optional, set to 0 if not required; sorted corresponding to ipMatchIndexes) *)
		fDissimilarityThreshold	:	LREAL;	(* Neglect irrelevant matches, i.e. dissimilarity > fDissimilarityThreshold *)
		eComparisonMethod	:	ETcVnContoursMatchComparisonMethod;	(* Method used for comparing the Hu moment invariants of the contours *)
		fAreaFactor	:	LREAL;	(* If > 0, the relative area difference between contours is scaled by this factor and added to the computed dissimilarity *)
		fAbsPositionFactor	:	LREAL;	(* If > 0, the absolute position difference between contours (i.e. the coordinates of the geometric contour centers) is scaled by this factor and added to the computed dissimilarity *)
		hrPrev	:	HRESULT;	(* HRESULT indicating the result of previous operations (If SUCCEEDED(hrPrev) equals false, no operation is executed.) *)
	END_VAR

END_FUNCTION

// Functions/Contour Analysis/F_VN_UprightBoundingRectangle

	{attribute 'TcIecLibraryType'}
	{attribute 'external_name' := 'F_VN_UprightBoundingRectangle_GUID_70206594_3F31_40FC_6B82_0DE89FC7E70C'}
	(* Determines the upright bounding rectangle of a set of points. *)
	FUNCTION F_VN_UprightBoundingRectangle : HRESULT
	VAR_INPUT
		ipPointSet	:	ITcVnContainer;	(* Source point set (ContainerType_Vector_TcVnPoint2_DINT or ContainerType_Vector_TcVnPoint2_REAL; The elements of this container are the individual points.) *)
		stRectangle	:	REFERENCE TO TcVnRectangle_UDINT;	(* Returns the determined rectangle *)
		hrPrev	:	HRESULT;	(* HRESULT indicating the result of previous operations (If SUCCEEDED(hrPrev) equals false, no operation is executed.) *)
	END_VAR

END_FUNCTION

// Functions/Image Filtering/F_VN_BilateralFilter

	{attribute 'TcIecLibraryType'}
	{attribute 'external_name' := 'F_VN_BilateralFilter_GUID_4BE06DF8_8A3E_41D1_67D8_E0AAD67C0016'}
	(* Apply a Bilateral filter to smooth the image but preserve edges. *)
	FUNCTION F_VN_BilateralFilter : HRESULT
	VAR_INPUT
		ipSrcImage	:	ITcVnImage;	(* Source image *)
		ipDestImage	:	REFERENCE TO ITcVnImage;	(* Destination image (Must be different from ipSrcImage! An appropriate destination image will be created if required.) *)
		nDiameter	:	DINT;	(* Diameter of the pixel neighborhood used for filtering (e.g. 5, 7, 9). If <= 0, it is automatically chosen dependend on fSigmaSpace. *)
		fSigmaColor	:	LREAL;	(* Sigma used for color space filtering (> 0). A larger value means that farther colors are mixed together. *)
		fSigmaSpace	:	LREAL;	(* Sigma used for coordinate space filtering (> 0). A larger value means that farther pixels can influence each other. *)
		hrPrev	:	HRESULT;	(* HRESULT indicating the result of previous operations (If SUCCEEDED(hrPrev) equals false, no operation is executed.) *)
	END_VAR

END_FUNCTION

// Functions/Image Filtering/F_VN_BilateralFilterExp

	{attribute 'TcIecLibraryType'}
	{attribute 'external_name' := 'F_VN_BilateralFilterExp_GUID_B7363814_02DA_477E_5ED7_0B5A6AB9F5D5'}
	(* Apply a Bilateral filter to smooth the image but preserve edges. (expert function) *)
	FUNCTION F_VN_BilateralFilterExp : HRESULT
	VAR_INPUT
		ipSrcImage	:	ITcVnImage;	(* Source image *)
		ipDestImage	:	REFERENCE TO ITcVnImage;	(* Destination image (Must be different from ipSrcImage! An appropriate destination image will be created if required.) *)
		nDiameter	:	DINT;	(* Diameter of the pixel neighborhood used for filtering (e.g. 5, 7, 9). If <= 0, it is automatically chosen dependend on fSigmaSpace. *)
		fSigmaColor	:	LREAL;	(* Sigma used for color space filtering (> 0). A larger value means that farther colors are mixed together. *)
		fSigmaSpace	:	LREAL;	(* Sigma used for coordinate space filtering (> 0). A larger value means that farther pixels can influence each other. *)
		eBorderType	:	ETcVnBorderInterpolationMethod;	(* Image border handling *)
		hrPrev	:	HRESULT;	(* HRESULT indicating the result of previous operations (If SUCCEEDED(hrPrev) equals false, no operation is executed.) *)
	END_VAR

END_FUNCTION

// Functions/Image Filtering/F_VN_BrightBorderObjects

	{attribute 'TcIecLibraryType'}
	{attribute 'external_name' := 'F_VN_BrightBorderObjects_GUID_AAEFE338_AA59_41B7_7B88_95FCA191CFD8'}
	(* Find bright objects connected to the image border within a gray-scale single-channel image. *)
	FUNCTION F_VN_BrightBorderObjects : HRESULT
	VAR_INPUT
		ipSrcImage	:	ITcVnImage;	(* Source image (USINT, UINT, INT, REAL, or LREAL, 1 channel) *)
		ipDestImage	:	REFERENCE TO ITcVnImage;	(* Destination image (An appropriate destination image will be created if required.) *)
		hrPrev	:	HRESULT;	(* HRESULT indicating the result of previous operations (If SUCCEEDED(hrPrev) equals false, no operation is executed.) *)
	END_VAR

END_FUNCTION

// Functions/Image Filtering/F_VN_CreateStructuringElement

	{attribute 'TcIecLibraryType'}
	{attribute 'external_name' := 'F_VN_CreateStructuringElement_GUID_883536F4_8118_4A7B_4357_7BA0E642FD4C'}
	(* Creates a structuring element for the usage with morphological operators and allocate an appropriate data buffer. The initial reference count is set to one if a new image interface is created and kept, otherwise. *)
	FUNCTION F_VN_CreateStructuringElement : HRESULT
	VAR_INPUT
		ipStructuringElement	:	REFERENCE TO ITcVnImage;	(* Returns the created structuring element (Non-zero interface pointers are reused.) *)
		eShape	:	ETcVnStructuringElementShape;	(* Shape of the structuring element (rectangle, cross, or ellipse) *)
		nWidth	:	UDINT;	(* Width *)
		nHeight	:	UDINT;	(* Height *)
		hrPrev	:	HRESULT;	(* HRESULT indicating the result of previous operations (If SUCCEEDED(hrPrev) equals false, no operation is executed.) *)
	END_VAR

END_FUNCTION

// Functions/Image Filtering/F_VN_CustomFilter

	{attribute 'TcIecLibraryType'}
	{attribute 'external_name' := 'F_VN_CustomFilter_GUID_6C782417_FFF9_4A20_60A6_CCEA32302913'}
	(* Apply a custom filter to the image. *)
	FUNCTION F_VN_CustomFilter : HRESULT
	VAR_INPUT
		ipSrcImage	:	ITcVnImage;	(* Source image *)
		ipDestImage	:	REFERENCE TO ITcVnImage;	(* Destination image (An appropriate destination image will be created if required.) *)
		eDestDepth	:	ETcVnElementType;	(* Destination image depth *)
		stKernel	:	REFERENCE TO TcVnMatrix;	(* Custom filter kernel with values of type REAL or LREAL *)
		hrPrev	:	HRESULT;	(* HRESULT indicating the result of previous operations (If SUCCEEDED(hrPrev) equals false, no operation is executed.) *)
	END_VAR

END_FUNCTION

// Functions/Image Filtering/F_VN_CustomFilterExp

	{attribute 'TcIecLibraryType'}
	{attribute 'external_name' := 'F_VN_CustomFilterExp_GUID_446F2DF9_D893_4845_57F3_7DDD6CA0BF81'}
	(* Apply a custom filter to the image. (expert function) *)
	FUNCTION F_VN_CustomFilterExp : HRESULT
	VAR_INPUT
		ipSrcImage	:	ITcVnImage;	(* Source image *)
		ipDestImage	:	REFERENCE TO ITcVnImage;	(* Destination image (An appropriate destination image will be created if required.) *)
		eDestDepth	:	ETcVnElementType;	(* Destination image depth *)
		stKernel	:	REFERENCE TO TcVnMatrix;	(* Custom filter kernel with values of type REAL or LREAL *)
		aAnchor	:	REFERENCE TO TcVnPoint;	(* Anchor point of the kernel *)
		fDelta	:	LREAL;	(* Value added to each pixel after filtering *)
		eBorderType	:	ETcVnBorderInterpolationMethod;	(* Image border handling *)
		hrPrev	:	HRESULT;	(* HRESULT indicating the result of previous operations (If SUCCEEDED(hrPrev) equals false, no operation is executed.) *)
	END_VAR

END_FUNCTION

// Functions/Image Filtering/F_VN_DarkBorderObjects

	{attribute 'TcIecLibraryType'}
	{attribute 'external_name' := 'F_VN_DarkBorderObjects_GUID_7F538751_7353_414C_77C6_8E876F10D196'}
	(* Find dark objects connected to the image border within a gray-scale single-channel image. (equivalent to filling holes) *)
	FUNCTION F_VN_DarkBorderObjects : HRESULT
	VAR_INPUT
		ipSrcImage	:	ITcVnImage;	(* Source image (USINT, UINT, INT, REAL, or LREAL, 1 channel) *)
		ipDestImage	:	REFERENCE TO ITcVnImage;	(* Destination image (An appropriate destination image will be created if required.) *)
		hrPrev	:	HRESULT;	(* HRESULT indicating the result of previous operations (If SUCCEEDED(hrPrev) equals false, no operation is executed.) *)
	END_VAR

END_FUNCTION

// Functions/Image Filtering/F_VN_FillHoles

	{attribute 'TcIecLibraryType'}
	{attribute 'external_name' := 'F_VN_FillHoles_GUID_1A242101_AA22_4DC1_4F1F_7C91CA2B8BB8'}
	(* Fill holes within a gray-scale single-channel image. (equivalent to finding dark border objects) *)
	FUNCTION F_VN_FillHoles : HRESULT
	VAR_INPUT
		ipSrcImage	:	ITcVnImage;	(* Source image (USINT, UINT, INT, REAL, or LREAL, 1 channel) *)
		ipDestImage	:	REFERENCE TO ITcVnImage;	(* Destination image (An appropriate destination image will be created if required.) *)
		hrPrev	:	HRESULT;	(* HRESULT indicating the result of previous operations (If SUCCEEDED(hrPrev) equals false, no operation is executed.) *)
	END_VAR

END_FUNCTION

// Functions/Image Filtering/F_VN_GaussianFilter

	{attribute 'TcIecLibraryType'}
	{attribute 'external_name' := 'F_VN_GaussianFilter_GUID_CA409851_82BC_40CC_6237_C89AD4958621'}
	(* Apply a Gaussian filter to smooth the image. *)
	FUNCTION F_VN_GaussianFilter : HRESULT
	VAR_INPUT
		ipSrcImage	:	ITcVnImage;	(* Source image *)
		ipDestImage	:	REFERENCE TO ITcVnImage;	(* Destination image (An appropriate destination image will be created if required.) *)
		nFilterWidth	:	UDINT;	(* Filter width in pixels (1, 3, 5, 7, ...) *)
		nFilterHeight	:	UDINT;	(* Filter height in pixels (1, 3, 5, 7, ...) *)
		hrPrev	:	HRESULT;	(* HRESULT indicating the result of previous operations (If SUCCEEDED(hrPrev) equals false, no operation is executed.) *)
	END_VAR

END_FUNCTION

// Functions/Image Filtering/F_VN_GaussianFilterExp

	{attribute 'TcIecLibraryType'}
	{attribute 'external_name' := 'F_VN_GaussianFilterExp_GUID_1B498EA4_FE3B_4485_617A_BF5586022CDF'}
	(* Apply a Gaussian filter to smooth the image. (expert function) *)
	FUNCTION F_VN_GaussianFilterExp : HRESULT
	VAR_INPUT
		ipSrcImage	:	ITcVnImage;	(* Source image *)
		ipDestImage	:	REFERENCE TO ITcVnImage;	(* Destination image (An appropriate destination image will be created if required.) *)
		nFilterWidth	:	UDINT;	(* Filter width in pixels (1, 3, 5, 7, ...) *)
		nFilterHeight	:	UDINT;	(* Filter height in pixels (1, 3, 5, 7, ...) *)
		fSigmaX	:	LREAL;	(* Gaussian kernel standard deviation in X direction (>= 0, automatically chosen if 0) *)
		fSigmaY	:	LREAL;	(* Gaussian kernel standard deviation in Y direction (>= 0, automatically chosen if 0) *)
		eBorderType	:	ETcVnBorderInterpolationMethod;	(* Image border handling *)
		hrPrev	:	HRESULT;	(* HRESULT indicating the result of previous operations (If SUCCEEDED(hrPrev) equals false, no operation is executed.) *)
	END_VAR

END_FUNCTION

// Functions/Image Filtering/F_VN_LaplacianFilter

	{attribute 'TcIecLibraryType'}
	{attribute 'external_name' := 'F_VN_LaplacianFilter_GUID_7D114857_C961_447A_59EF_0085E2A215E2'}
	(* Apply a Laplacian filter to an image. *)
	FUNCTION F_VN_LaplacianFilter : HRESULT
	VAR_INPUT
		ipSrcImage	:	ITcVnImage;	(* Source image *)
		ipDestImage	:	REFERENCE TO ITcVnImage;	(* Destination image (An appropriate destination image will be created if required.) *)
		eDestDepth	:	ETcVnElementType;	(* Destination image depth *)
		hrPrev	:	HRESULT;	(* HRESULT indicating the result of previous operations (If SUCCEEDED(hrPrev) equals false, no operation is executed.) *)
	END_VAR

END_FUNCTION

// Functions/Image Filtering/F_VN_LaplacianFilterExp

	{attribute 'TcIecLibraryType'}
	{attribute 'external_name' := 'F_VN_LaplacianFilterExp_GUID_DF2787EA_8B8A_4126_5EF9_8CC89EFBA64F'}
	(* Apply a Laplacian filter to an image. (expert function) *)
	FUNCTION F_VN_LaplacianFilterExp : HRESULT
	VAR_INPUT
		ipSrcImage	:	ITcVnImage;	(* Source image *)
		ipDestImage	:	REFERENCE TO ITcVnImage;	(* Destination image (An appropriate destination image will be created if required.) *)
		eDestDepth	:	ETcVnElementType;	(* Destination image depth *)
		nKernelSize	:	UDINT;	(* Aperture size used to compute the second-derivative filters (1, 3, 5, ..., 31) *)
		fScale	:	LREAL;	(* Scale factor for the computed derivative values *)
		fDelta	:	LREAL;	(* Delta value that is added to the results before storing them *)
		eBorderType	:	ETcVnBorderInterpolationMethod;	(* Image border handling *)
		hrPrev	:	HRESULT;	(* HRESULT indicating the result of previous operations (If SUCCEEDED(hrPrev) equals false, no operation is executed.) *)
	END_VAR

END_FUNCTION

// Functions/Image Filtering/F_VN_LocalMaxima

	{attribute 'TcIecLibraryType'}
	{attribute 'external_name' := 'F_VN_LocalMaxima_GUID_5C9B6CF3_C33E_4944_6415_F920DFFDFE5F'}
	(* Find local maxima in a gray-scale single-channel image. The found maxima are marked by a value of 1 in the destination image. *)
	FUNCTION F_VN_LocalMaxima : HRESULT
	VAR_INPUT
		ipSrcImage	:	ITcVnImage;	(* Source image (USINT or UINT, 1 channel) *)
		ipDestImage	:	REFERENCE TO ITcVnImage;	(* Destination image (An appropriate destination image will be created if required.) *)
		hrPrev	:	HRESULT;	(* HRESULT indicating the result of previous operations (If SUCCEEDED(hrPrev) equals false, no operation is executed.) *)
	END_VAR

END_FUNCTION

// Functions/Image Filtering/F_VN_LocalMinima

	{attribute 'TcIecLibraryType'}
	{attribute 'external_name' := 'F_VN_LocalMinima_GUID_6CCB026E_58BC_42D4_74D8_74350EB83EB0'}
	(* Find local minima in a gray-scale single-channel image. The found minima are marked by a value of 1 in the destination image. *)
	FUNCTION F_VN_LocalMinima : HRESULT
	VAR_INPUT
		ipSrcImage	:	ITcVnImage;	(* Source image (USINT or UINT, 1 channel) *)
		ipDestImage	:	REFERENCE TO ITcVnImage;	(* Destination image (An appropriate destination image will be created if required.) *)
		hrPrev	:	HRESULT;	(* HRESULT indicating the result of previous operations (If SUCCEEDED(hrPrev) equals false, no operation is executed.) *)
	END_VAR

END_FUNCTION

// Functions/Image Filtering/F_VN_MedianFilter

	{attribute 'TcIecLibraryType'}
	{attribute 'external_name' := 'F_VN_MedianFilter_GUID_47D81315_C0DF_4934_6F7F_EBE4C13057F8'}
	(* Apply a Median filter to an image. *)
	FUNCTION F_VN_MedianFilter : HRESULT
	VAR_INPUT
		ipSrcImage	:	ITcVnImage;	(* Source image (for nFilterSize 3 or 5: USINT, UINT, REAL. For bigger filters, only USINT is supported. *)
		ipDestImage	:	REFERENCE TO ITcVnImage;	(* Destination image (An appropriate destination image will be created if required.) *)
		nFilterSize	:	UDINT;	(* Size (width and height) of the filter (3, 5, 7, ...) *)
		hrPrev	:	HRESULT;	(* HRESULT indicating the result of previous operations (If SUCCEEDED(hrPrev) equals false, no operation is executed.) *)
	END_VAR

END_FUNCTION

// Functions/Image Filtering/F_VN_MorphologicalOperator

	{attribute 'TcIecLibraryType'}
	{attribute 'external_name' := 'F_VN_MorphologicalOperator_GUID_EDD30F65_A28E_44E6_43F2_4AA38453E57F'}
	(* Apply a morphological operator. *)
	FUNCTION F_VN_MorphologicalOperator : HRESULT
	VAR_INPUT
		ipSrcImage	:	ITcVnImage;	(* Source image *)
		ipDestImage	:	REFERENCE TO ITcVnImage;	(* Destination image (An appropriate destination image will be created if required.) *)
		eOperator	:	ETcVnMorphologicalOperator;	(* Operator type *)
		ipStructuringElement	:	ITcVnImage;	(* Structuring element to be applied (Typically created via F_VN_CreateStructuringElement.) *)
		hrPrev	:	HRESULT;	(* HRESULT indicating the result of previous operations (If SUCCEEDED(hrPrev) equals false, no operation is executed.) *)
	END_VAR

END_FUNCTION

// Functions/Image Filtering/F_VN_RemoveLocalMaxima

	{attribute 'TcIecLibraryType'}
	{attribute 'external_name' := 'F_VN_RemoveLocalMaxima_GUID_3C429603_F72B_41E1_434D_B8E8A83BB2DF'}
	(* Remove local maxima up to a given height from a gray-scale single-channel image. *)
	FUNCTION F_VN_RemoveLocalMaxima : HRESULT
	VAR_INPUT
		ipSrcImage	:	ITcVnImage;	(* Source image (USINT, UINT, INT, REAL, or LREAL, 1 channel) *)
		ipDestImage	:	REFERENCE TO ITcVnImage;	(* Destination image (An appropriate destination image will be created if required.) *)
		fHeight	:	LREAL;	(* Maximum height of the maxima to be removed (must be greater than 0) *)
		hrPrev	:	HRESULT;	(* HRESULT indicating the result of previous operations (If SUCCEEDED(hrPrev) equals false, no operation is executed.) *)
	END_VAR

END_FUNCTION

// Functions/Image Filtering/F_VN_RemoveLocalMinima

	{attribute 'TcIecLibraryType'}
	{attribute 'external_name' := 'F_VN_RemoveLocalMinima_GUID_8AED91A0_925B_4A69_76B3_5B7C8861E5BF'}
	(* Remove local minima up to a given height from a gray-scale single-channel image. *)
	FUNCTION F_VN_RemoveLocalMinima : HRESULT
	VAR_INPUT
		ipSrcImage	:	ITcVnImage;	(* Source image (USINT, UINT, INT, REAL, or LREAL, 1 channel) *)
		ipDestImage	:	REFERENCE TO ITcVnImage;	(* Destination image (An appropriate destination image will be created if required.) *)
		fHeight	:	LREAL;	(* Maximum height of the minima to be removed (must be greater than 0) *)
		hrPrev	:	HRESULT;	(* HRESULT indicating the result of previous operations (If SUCCEEDED(hrPrev) equals false, no operation is executed.) *)
	END_VAR

END_FUNCTION

// Functions/Image Filtering/F_VN_ScharrFilter

	{attribute 'TcIecLibraryType'}
	{attribute 'external_name' := 'F_VN_ScharrFilter_GUID_13AD7402_EFDE_4CAE_6DB0_6C0CA3018923'}
	(* Calculates the first order derivative in x or y direction using a Scharr filter. *)
	FUNCTION F_VN_ScharrFilter : HRESULT
	VAR_INPUT
		ipSrcImage	:	ITcVnImage;	(* Source image *)
		ipDestImage	:	REFERENCE TO ITcVnImage;	(* Destination image (An appropriate destination image will be created if required.) *)
		eDestDepth	:	ETcVnElementType;	(* Destination image depth *)
		eFilterDirection	:	ETcVnFilterDirection;	(* Filter direction *)
		hrPrev	:	HRESULT;	(* HRESULT indicating the result of previous operations (If SUCCEEDED(hrPrev) equals false, no operation is executed.) *)
	END_VAR

END_FUNCTION

// Functions/Image Filtering/F_VN_ScharrFilterExp

	{attribute 'TcIecLibraryType'}
	{attribute 'external_name' := 'F_VN_ScharrFilterExp_GUID_3BEF9604_89A8_4747_69BB_744D33490B0B'}
	(* Calculates the first order derivative in x or y direction using a Scharr filter. (expert function) *)
	FUNCTION F_VN_ScharrFilterExp : HRESULT
	VAR_INPUT
		ipSrcImage	:	ITcVnImage;	(* Source image *)
		ipDestImage	:	REFERENCE TO ITcVnImage;	(* Destination image (An appropriate destination image will be created if required.) *)
		eDestDepth	:	ETcVnElementType;	(* Destination image depth *)
		eFilterDirection	:	ETcVnFilterDirection;	(* Filter direction *)
		fScale	:	LREAL;	(* Scale factor for the computed derivative values *)
		fDelta	:	LREAL;	(* Delta value that is added to the results prior to storing them in dest *)
		eBorderType	:	ETcVnBorderInterpolationMethod;	(* Image border handling *)
		hrPrev	:	HRESULT;	(* HRESULT indicating the result of previous operations (If SUCCEEDED(hrPrev) equals false, no operation is executed.) *)
	END_VAR

END_FUNCTION

// Functions/Image Filtering/F_VN_SeparableCustomFilter

	{attribute 'TcIecLibraryType'}
	{attribute 'external_name' := 'F_VN_SeparableCustomFilter_GUID_4CF7E46F_947F_4E09_4F79_7BAF5EC2EB59'}
	(* Apply a separable custom filter to the image. *)
	FUNCTION F_VN_SeparableCustomFilter : HRESULT
	VAR_INPUT
		ipSrcImage	:	ITcVnImage;	(* Source image *)
		ipDestImage	:	REFERENCE TO ITcVnImage;	(* Destination image (An appropriate destination image will be created if required.) *)
		eDestDepth	:	ETcVnElementType;	(* Destination image depth *)
		stKernelX	:	REFERENCE TO TcVnMatrix;	(* 1D custom row-filter kernel with values of type REAL or LREAL *)
		stKernelY	:	REFERENCE TO TcVnMatrix;	(* 1D custom column-filter kernel with values of type REAL or LREAL *)
		hrPrev	:	HRESULT;	(* HRESULT indicating the result of previous operations (If SUCCEEDED(hrPrev) equals false, no operation is executed.) *)
	END_VAR

END_FUNCTION

// Functions/Image Filtering/F_VN_SeparableCustomFilterExp

	{attribute 'TcIecLibraryType'}
	{attribute 'external_name' := 'F_VN_SeparableCustomFilterExp_GUID_E323CAF5_95AE_4C9D_6461_0F80FFF767A7'}
	(* Apply a separable custom filter to the image. (expert function) *)
	FUNCTION F_VN_SeparableCustomFilterExp : HRESULT
	VAR_INPUT
		ipSrcImage	:	ITcVnImage;	(* Source image *)
		ipDestImage	:	REFERENCE TO ITcVnImage;	(* Destination image (An appropriate destination image will be created if required.) *)
		eDestDepth	:	ETcVnElementType;	(* Destination image depth *)
		stKernelX	:	REFERENCE TO TcVnMatrix;	(* 1D custom row-filter kernel with values of type REAL or LREAL *)
		stKernelY	:	REFERENCE TO TcVnMatrix;	(* 1D custom column-filter kernel with values of type REAL or LREAL *)
		aAnchor	:	REFERENCE TO TcVnPoint;	(* Anchor point of the kernel *)
		fDelta	:	LREAL;	(* Value added to each pixel after filtering *)
		eBorderType	:	ETcVnBorderInterpolationMethod;	(* Image border handling *)
		hrPrev	:	HRESULT;	(* HRESULT indicating the result of previous operations (If SUCCEEDED(hrPrev) equals false, no operation is executed.) *)
	END_VAR

END_FUNCTION

// Functions/Image Filtering/F_VN_SobelFilter

	{attribute 'TcIecLibraryType'}
	{attribute 'external_name' := 'F_VN_SobelFilter_GUID_57CE5A32_6BB6_46B2_6D4C_9805BAB50E6C'}
	(* Calculates the first, second, or mixed image derivatives using an extended Sobel filter. *)
	FUNCTION F_VN_SobelFilter : HRESULT
	VAR_INPUT
		ipSrcImage	:	ITcVnImage;	(* Source image *)
		ipDestImage	:	REFERENCE TO ITcVnImage;	(* Destination image (An appropriate destination image will be created if required.) *)
		eDestDepth	:	ETcVnElementType;	(* Destination image depth *)
		nXOrder	:	UDINT;	(* Order of the x-derivative (0, 1, 2) *)
		nYOrder	:	UDINT;	(* Order of the y-derivative (0, 1, 2) *)
		hrPrev	:	HRESULT;	(* HRESULT indicating the result of previous operations (If SUCCEEDED(hrPrev) equals false, no operation is executed.) *)
	END_VAR

END_FUNCTION

// Functions/Image Filtering/F_VN_SobelFilterExp

	{attribute 'TcIecLibraryType'}
	{attribute 'external_name' := 'F_VN_SobelFilterExp_GUID_D4A6716E_00CF_4B2D_4652_AFA25B1F80DB'}
	(* Calculates the first, second, third, or mixed image derivatives using an extended Sobel filter. (expert function) *)
	FUNCTION F_VN_SobelFilterExp : HRESULT
	VAR_INPUT
		ipSrcImage	:	ITcVnImage;	(* Source image *)
		ipDestImage	:	REFERENCE TO ITcVnImage;	(* Destination image (An appropriate destination image will be created if required.) *)
		eDestDepth	:	ETcVnElementType;	(* Destination image depth *)
		nXOrder	:	UDINT;	(* Order of the x-derivative (must be < nKernelSize) *)
		nYOrder	:	UDINT;	(* Order of the y-derivative (must be < nKernelSize) *)
		nKernelSize	:	UDINT;	(* Size of the extended Sobel kernel (3, 5, 7, ..., 31) *)
		fScale	:	LREAL;	(* Scale factor for the computed derivative values *)
		fDelta	:	LREAL;	(* Delta value that is added to the results prior to storing them in dest *)
		eBorderType	:	ETcVnBorderInterpolationMethod;	(* Image border handling *)
		hrPrev	:	HRESULT;	(* HRESULT indicating the result of previous operations (If SUCCEEDED(hrPrev) equals false, no operation is executed.) *)
	END_VAR

END_FUNCTION

// Functions/Miscellaneous/F_VN_ClipLineToBoundary

	{attribute 'TcIecLibraryType'}
	{attribute 'external_name' := 'F_VN_ClipLineToBoundary_GUID_EB658276_C4D3_4EA2_6B36_4FB748A4C67D'}
	(* Clips a line to a rectangular boundary. *)
	FUNCTION F_VN_ClipLineToBoundary : HRESULT
	VAR_INPUT
		aLine	:	REFERENCE TO TcVnVector4_LREAL;	(* The first and second element describe the x and y component of the direction vector. The third and fourth element describe the x and y component of the position vector. *)
		nX1	:	DINT;	(* x of top left rectangle point *)
		nY1	:	DINT;	(* y of top left rectangle point *)
		nX2	:	DINT;	(* x of bottom right rectangle point *)
		nY2	:	DINT;	(* Y of bottom right rectangle point *)
		aStartPoint	:	REFERENCE TO TcVnPoint2_REAL;	(* Returns the clipped starting point of the line. *)
		aEndPoint	:	REFERENCE TO TcVnPoint2_REAL;	(* Returns the clipped end point of the line. *)
		hrPrev	:	HRESULT;	(* HRESULT indicating the result of previous operations (If SUCCEEDED(hrPrev) equals false, no operation is executed.) *)
	END_VAR

END_FUNCTION

// Functions/Miscellaneous/F_VN_ClipLineToBoundary_ITcVnImage

	{attribute 'TcIecLibraryType'}
	{attribute 'external_name' := 'F_VN_ClipLineToBoundary_ITcVnImage_GUID_502D1086_C675_4921_71A3_FD3336969F8B'}
	(* Clips a line to the boundary of an image. *)
	FUNCTION F_VN_ClipLineToBoundary_ITcVnImage : HRESULT
	VAR_INPUT
		aLine	:	REFERENCE TO TcVnVector4_LREAL;	(* The first and second element describe the x and y component of the direction vector. The third and fourth element describe the x and y component of the position vector. *)
		ipImage	:	ITcVnImage;	(* Image, from which to derive the boundary *)
		aStartPoint	:	REFERENCE TO TcVnPoint2_REAL;	(* Returns the clipped starting point of the line. *)
		aEndPoint	:	REFERENCE TO TcVnPoint2_REAL;	(* Returns the clipped end point of the line. *)
		hrPrev	:	HRESULT;	(* HRESULT indicating the result of previous operations (If SUCCEEDED(hrPrev) equals false, no operation is executed.) *)
	END_VAR

END_FUNCTION

// Functions/Miscellaneous/F_VN_ClipLineToBoundary_TcVnRectangle_DINT

	{attribute 'TcIecLibraryType'}
	{attribute 'external_name' := 'F_VN_ClipLineToBoundary_TcVnRectangle_DINT_GUID_33EDADFF_5A06_4852_6556_CC5B82D1EFE8'}
	(* Clips a line to a rectangular boundary. *)
	FUNCTION F_VN_ClipLineToBoundary_TcVnRectangle_DINT : HRESULT
	VAR_INPUT
		aLine	:	REFERENCE TO TcVnVector4_LREAL;	(* The first and second element describe the x and y component of the direction vector. The third and fourth element describe the x and y component of the position vector. *)
		stRectangle	:	REFERENCE TO TcVnRectangle_DINT;	(* Rectangular boundary *)
		aStartPoint	:	REFERENCE TO TcVnPoint2_REAL;	(* Returns the clipped starting point of the line. *)
		aEndPoint	:	REFERENCE TO TcVnPoint2_REAL;	(* Returns the clipped end point of the line. *)
		hrPrev	:	HRESULT;	(* HRESULT indicating the result of previous operations (If SUCCEEDED(hrPrev) equals false, no operation is executed.) *)
	END_VAR

END_FUNCTION

// Functions/Miscellaneous/F_VN_HuMomentInvariants

	{attribute 'TcIecLibraryType'}
	{attribute 'external_name' := 'F_VN_HuMomentInvariants_GUID_0868EACA_6C27_4649_5304_0E3EE0030D2B'}
	(* Computes the Hu moment invariants. *)
	FUNCTION F_VN_HuMomentInvariants : HRESULT
	VAR_INPUT
		stMoments	:	REFERENCE TO TcVnMoments;	(* Moments from which to compute the Hu invariants *)
		aHuInvariants	:	REFERENCE TO TcVnArray7_LREAL;	(* Returns the Hu moment invariants *)
		hrPrev	:	HRESULT;	(* HRESULT indicating the result of previous operations (If SUCCEEDED(hrPrev) equals false, no operation is executed.) *)
	END_VAR

END_FUNCTION

// Functions/Miscellaneous/F_VN_InitMatrixStruct

	{attribute 'TcIecLibraryType'}
	{attribute 'external_name' := 'F_VN_InitMatrixStruct_GUID_33702A96_58A2_4704_54C5_3A8BF0EA3D81'}
	(* Initialize a struct of the type TcVnMatrix extending a buffer with metainformation so that it can be used as a matrix. *)
	FUNCTION F_VN_InitMatrixStruct : HRESULT
	VAR_INPUT
		pSrcBuffer	:	PVOID;	(* Source buffer *)
		stDestMatrix	:	REFERENCE TO TcVnMatrix;	(* Returns completed matrix struct *)
		nRows	:	UDINT;	(* Matrix rows *)
		nCols	:	UDINT;	(* Matrix columns *)
		eElementType	:	ETcVnElementType;	(* Type of the matrix elements *)
		hrPrev	:	HRESULT;	(* HRESULT indicating the result of previous operations (If SUCCEEDED(hrPrev) equals false, no operation is executed.) *)
	END_VAR

END_FUNCTION

// Functions/Miscellaneous/F_VN_InvertMatrix3x3

	{attribute 'TcIecLibraryType'}
	{attribute 'external_name' := 'F_VN_InvertMatrix3x3_GUID_5C49241D_6140_403D_6C4A_9790EBD59D60'}
	(* Invert a 3x3 matrix. *)
	FUNCTION F_VN_InvertMatrix3x3 : HRESULT
	VAR_INPUT
		aSrcMatrix	:	REFERENCE TO TcVnMatrix3x3_LREAL;	(* Source matrix *)
		aInvertedMatrix	:	REFERENCE TO TcVnMatrix3x3_LREAL;	(* Returns inverted matrix *)
		hrPrev	:	HRESULT;	(* HRESULT indicating the result of previous operations (If SUCCEEDED(hrPrev) equals false, no operation is executed.) *)
	END_VAR

END_FUNCTION

// Functions/Miscellaneous/F_VN_LineIntersectionPoint

	{attribute 'TcIecLibraryType'}
	{attribute 'external_name' := 'F_VN_LineIntersectionPoint_GUID_BD268DC7_44B4_43CE_5BED_BD4EB0BE3015'}
	(* Computes the intersection point between two lines (returns S_FALSE if the provided lines are parallel). *)
	FUNCTION F_VN_LineIntersectionPoint : HRESULT
	VAR_INPUT
		aLine1	:	REFERENCE TO TcVnVector4_LREAL;	(* First line. The first and second element describe the x and y component of a vector collinear to the line. The third and fourth element describe the x and y component of a point on the line. *)
		aLine2	:	REFERENCE TO TcVnVector4_LREAL;	(* Second line. The first and second element describe the x and y component of a vector collinear to the line. The third and fourth element describe the x and y component of a point on the line. *)
		aIntersecPoint	:	REFERENCE TO TcVnPoint2_REAL;	(* Returns the intersection point of aLine1 and aLine2. *)
		hrPrev	:	HRESULT;	(* HRESULT indicating the result of previous operations (If SUCCEEDED(hrPrev) equals false, no operation is executed.) *)
	END_VAR

END_FUNCTION

// Functions/Miscellaneous/F_VN_LineIntersectionPointAndAngle

	{attribute 'TcIecLibraryType'}
	{attribute 'external_name' := 'F_VN_LineIntersectionPointAndAngle_GUID_B65473E1_3E0B_421B_5CCC_43C8C7EAE42C'}
	(* Computes the intersection point and angle between two lines (returns S_FALSE if the provided lines are parallel). *)
	FUNCTION F_VN_LineIntersectionPointAndAngle : HRESULT
	VAR_INPUT
		aLine1	:	REFERENCE TO TcVnVector4_LREAL;	(* First line. The first and second element describe the x and y component of a vector collinear to the line. The third and fourth element describe the x and y component of a point on the line. *)
		aLine2	:	REFERENCE TO TcVnVector4_LREAL;	(* Second line. The first and second element describe the x and y component of a vector collinear to the line. The third and fourth element describe the x and y component of a point on the line. *)
		aIntersecPoint	:	REFERENCE TO TcVnPoint2_REAL;	(* Returns the intersection point of aLine1 and aLine2. *)
		fAngle	:	REFERENCE TO REAL;	(* Returns the intersection angle of aLine1 and aLine2. *)
		bAngleInDegrees	:	BOOL;	(* If TRUE, fAngle is in degrees. If FALSE, fAngle is in radians. *)
		hrPrev	:	HRESULT;	(* HRESULT indicating the result of previous operations (If SUCCEEDED(hrPrev) equals false, no operation is executed.) *)
	END_VAR

END_FUNCTION

// Functions/Miscellaneous/F_VN_MultiplyMatrices

	{attribute 'TcIecLibraryType'}
	{attribute 'external_name' := 'F_VN_MultiplyMatrices_GUID_5AA3721E_513B_4002_589A_9D0FDE905CA9'}
	(* Matrix multiplication of two matrices (A * B = C). All matrices are represented by structs holding a pointer to an array of the appropriate size. *)
	FUNCTION F_VN_MultiplyMatrices : HRESULT
	VAR_INPUT
		stSrcMatrix1	:	REFERENCE TO TcVnMatrix;	(* First source matrix (A) *)
		stSrcMatrix2	:	REFERENCE TO TcVnMatrix;	(* Second source matrix (B) *)
		stDestMatrix	:	REFERENCE TO TcVnMatrix;	(* Destination matrix (C) (The destination matrix is filled by this function, but the required memory needs to be provided.) *)
		hrPrev	:	HRESULT;	(* HRESULT indicating the result of previous operations (If SUCCEEDED(hrPrev) equals false, no operation is executed.) *)
	END_VAR

END_FUNCTION

// Functions/Basic Image Operations/F_VN_CombineImageChannels

	{attribute 'TcIecLibraryType'}
	{attribute 'external_name' := 'F_VN_CombineImageChannels_GUID_7A3D00D8_5932_4C2C_47EC_0EB4F1EC8BEC'}
	(* Combines several single-channel images into one multi-channel image. *)
	FUNCTION F_VN_CombineImageChannels : HRESULT
	VAR_INPUT
		pSrcImages	:	PVOID;	(* Pointer to an array of single-channel source images *)
		ipDestImage	:	REFERENCE TO ITcVnImage;	(* Multi-channel destination image (An appropriate destination image will be created if required.) *)
		nSrcArraySize	:	UINT;	(* pSrcImages array size *)
		hrPrev	:	HRESULT;	(* HRESULT indicating the result of previous operations (If SUCCEEDED(hrPrev) equals false, no operation is executed.) *)
	END_VAR

END_FUNCTION

// Functions/Basic Image Operations/F_VN_ConvertElementType

	{attribute 'TcIecLibraryType'}
	{attribute 'external_name' := 'F_VN_ConvertElementType_GUID_DB87FB3B_B67B_459C_6C55_54CF581D3B88'}
	(* Converts an image to another element type. *)
	FUNCTION F_VN_ConvertElementType : HRESULT
	VAR_INPUT
		ipSrcImage	:	ITcVnImage;	(* Source image *)
		ipDestImage	:	REFERENCE TO ITcVnImage;	(* Destination image (An appropriate destination image will be created if required.) *)
		eElementType	:	ETcVnElementType;	(* Desired element type of the destination image *)
		hrPrev	:	HRESULT;	(* HRESULT indicating the result of previous operations (If SUCCEEDED(hrPrev) equals false, no operation is executed.) *)
	END_VAR

END_FUNCTION

// Functions/Basic Image Operations/F_VN_ConvertElementTypeExp

	{attribute 'TcIecLibraryType'}
	{attribute 'external_name' := 'F_VN_ConvertElementTypeExp_GUID_2B706411_D717_4961_754C_4ECD1B0127D3'}
	(* Converts an image to another element type. (expert function) *)
	FUNCTION F_VN_ConvertElementTypeExp : HRESULT
	VAR_INPUT
		ipSrcImage	:	ITcVnImage;	(* Source image *)
		ipDestImage	:	REFERENCE TO ITcVnImage;	(* Destination image (An appropriate destination image will be created if required.) *)
		eElementType	:	ETcVnElementType;	(* Desired element type of the destination image *)
		fScaleFactor	:	LREAL;	(* Scale factor for the pixel values *)
		fDelta	:	LREAL;	(* Value that is added to the scaled pixel values *)
		hrPrev	:	HRESULT;	(* HRESULT indicating the result of previous operations (If SUCCEEDED(hrPrev) equals false, no operation is executed.) *)
	END_VAR

END_FUNCTION

// Functions/Basic Image Operations/F_VN_CopyImage

	{attribute 'TcIecLibraryType'}
	{attribute 'external_name' := 'F_VN_CopyImage_GUID_8528176A_E1C2_4CEE_5F9D_2978A7D83010'}
	(* Creates a deep copy of an image. *)
	FUNCTION F_VN_CopyImage : HRESULT
	VAR_INPUT
		ipSrcImage	:	ITcVnImage;	(* Source image *)
		ipDestImage	:	REFERENCE TO ITcVnImage;	(* Destination image (An appropriate destination image will be created if required.) *)
		hrPrev	:	HRESULT;	(* HRESULT indicating the result of previous operations (If SUCCEEDED(hrPrev) equals false, no operation is executed.) *)
	END_VAR

END_FUNCTION

// Functions/Basic Image Operations/F_VN_CopyImageRegion

	{attribute 'TcIecLibraryType'}
	{attribute 'external_name' := 'F_VN_CopyImageRegion_GUID_BC187631_FED7_4E32_6C55_CEFDE80685BF'}
	(* Deep copy the specified region of interest into a new image. *)
	FUNCTION F_VN_CopyImageRegion : HRESULT
	VAR_INPUT
		ipSrcImage	:	ITcVnImage;	(* Source image *)
		nX	:	UDINT;	(* Left boundary (inclusive 0-based index) *)
		nY	:	UDINT;	(* Upper boundary (inclusive 0-based index) *)
		nWidth	:	UDINT;	(* ROI width *)
		nHeight	:	UDINT;	(* ROI height *)
		ipDestImage	:	REFERENCE TO ITcVnImage;	(* Destination image (An appropriate destination image will be created if required.) *)
		hrPrev	:	HRESULT;	(* HRESULT indicating the result of previous operations (If SUCCEEDED(hrPrev) equals false, no operation is executed.) *)
	END_VAR

END_FUNCTION

// Functions/Basic Image Operations/F_VN_CopyImageRegionToRegion

	{attribute 'TcIecLibraryType'}
	{attribute 'external_name' := 'F_VN_CopyImageRegionToRegion_GUID_2B377BB5_A27C_4C83_4676_DD4B173CE5C5'}
	(* Copy an image region into another image region. *)
	FUNCTION F_VN_CopyImageRegionToRegion : HRESULT
	VAR_INPUT
		ipSrcImage	:	ITcVnImage;	(* Source image *)
		nXSrc	:	UDINT;	(* Left boundary in ipSrcImage (inclusive 0-based index) *)
		nYSrc	:	UDINT;	(* Upper boundary in ipSrcImage (inclusive 0-based index) *)
		nWidth	:	UDINT;	(* ROI width *)
		nHeight	:	UDINT;	(* ROI height *)
		ipDestImage	:	ITcVnImage;	(* Destination image (same type as ipSrcImage) *)
		nXDest	:	UDINT;	(* Left boundary in ipDestImage (inclusive 0-based index) *)
		nYDest	:	UDINT;	(* Upper boundary in ipDestImage (inclusive 0-based index) *)
		hrPrev	:	HRESULT;	(* HRESULT indicating the result of previous operations (If SUCCEEDED(hrPrev) equals false, no operation is executed.) *)
	END_VAR

END_FUNCTION

// Functions/Basic Image Operations/F_VN_CopyIntoDisplayableImage

	{attribute 'TcIecLibraryType'}
	{attribute 'external_name' := 'F_VN_CopyIntoDisplayableImage_GUID_2FA25F46_93CF_4FB0_5AB3_65D8155CFCA9'}
	(* Copys an image into a displayable image. If you do not want to use ipSrcImage after this function call, you might want to use F_VN_TransformIntoDisplayableImage instead for better performance. *)
	FUNCTION F_VN_CopyIntoDisplayableImage : HRESULT
	VAR_INPUT
		ipSrcImage	:	ITcVnImage;	(* Source image *)
		ipDestImage	:	REFERENCE TO ITcVnDisplayableImage;	(* Returns the displayable image *)
		hrPrev	:	HRESULT;	(* HRESULT indicating the result of previous operations (If SUCCEEDED(hrPrev) equals false, no operation is executed.) *)
	END_VAR

END_FUNCTION

// Functions/Basic Image Operations/F_VN_TransformIntoDisplayableImage

	{attribute 'TcIecLibraryType'}
	{attribute 'external_name' := 'F_VN_TransformIntoDisplayableImage_GUID_DE2CC749_C9E5_4C90_4DDD_1AA68E70FA1C'}
	(* Transform an image into a displayable image. The source image will be released and zeroed while existing destination images will be released and overwritten with the function result. The source image must not be used anywhere else and the transformation is very fast. If you want to use ipSrcImage after this function call, use F_VN_CopyIntoDisplayableImage instead. *)
	FUNCTION F_VN_TransformIntoDisplayableImage : HRESULT
	VAR_INPUT
		ipSrcImage	:	REFERENCE TO ITcVnImage;	(* Source image *)
		ipDestImage	:	REFERENCE TO ITcVnDisplayableImage;	(* Returns the displayable image *)
		hrPrev	:	HRESULT;	(* HRESULT indicating the result of previous operations (If SUCCEEDED(hrPrev) equals false, no operation is executed.) *)
	END_VAR

END_FUNCTION

// Functions/Basic Image Operations/F_VN_CreateAssociatedImage

	{attribute 'TcIecLibraryType'}
	{attribute 'external_name' := 'F_VN_CreateAssociatedImage_GUID_9C1F95A1_2985_4DD2_7894_7E7B74423737'}
	(* Creates a new image that shares its data with the source image. E.g. useful to work on different (disjoint) ROIs in parallel. *)
	FUNCTION F_VN_CreateAssociatedImage : HRESULT
	VAR_INPUT
		ipSrcImage	:	ITcVnImage;	(* Source image *)
		ipDestImage	:	REFERENCE TO ITcVnImage;	(* Returns the created image (Non-zero interface pointers are reused.) *)
		hrPrev	:	HRESULT;	(* HRESULT indicating the result of previous operations (If SUCCEEDED(hrPrev) equals false, no operation is executed.) *)
	END_VAR

END_FUNCTION

// Functions/Basic Image Operations/F_VN_CreateEmptyImage

	{attribute 'TcIecLibraryType'}
	{attribute 'external_name' := 'F_VN_CreateEmptyImage_GUID_5B120016_A80C_4DA3_47B3_991D20065844'}
	(* Creates an empty image without allocating any data buffer. The initial reference count is set to one if a new image interface is created and kept, otherwise. *)
	FUNCTION F_VN_CreateEmptyImage : HRESULT
	VAR_INPUT
		ipImage	:	REFERENCE TO ITcVnImage;	(* Returns the created image *)
		hrPrev	:	HRESULT;	(* HRESULT indicating the result of previous operations (If SUCCEEDED(hrPrev) equals false, no operation is executed.) *)
	END_VAR

END_FUNCTION

// Functions/Basic Image Operations/F_VN_CreateImage

	{attribute 'TcIecLibraryType'}
	{attribute 'external_name' := 'F_VN_CreateImage_GUID_51B807DC_6A5C_4543_71CC_1101C37E503F'}
	(* Creates an image and allocate an appropriate data buffer. The initial reference count is set to one if a new image interface is created and kept, otherwise. *)
	FUNCTION F_VN_CreateImage : HRESULT
	VAR_INPUT
		ipImage	:	REFERENCE TO ITcVnImage;	(* Returns the created image (Non-zero interface pointers are reused.) *)
		nWidth	:	UDINT;	(* Image width *)
		nHeight	:	UDINT;	(* Image height *)
		ePixelType	:	ETcVnElementType;	(* Pixel type *)
		nChannelNum	:	UDINT;	(* Number of channels (1 to 255) *)
		hrPrev	:	HRESULT;	(* HRESULT indicating the result of previous operations (If SUCCEEDED(hrPrev) equals false, no operation is executed.) *)
	END_VAR

END_FUNCTION

// Functions/Basic Image Operations/F_VN_CreateImageFromArray

	{attribute 'TcIecLibraryType'}
	{attribute 'external_name' := 'F_VN_CreateImageFromArray_GUID_BD01FA3F_146A_4026_71FB_DD7B0D997C59'}
	(* Creates an image and initialize it with the provided data. The initial reference count is set to one if a new image interface is created and kept, otherwise. *)
	FUNCTION F_VN_CreateImageFromArray : HRESULT
	VAR_INPUT
		pData	:	PVOID;	(* Pointer to the 1D data array. Make sure that the array contains at least nWidth * nHeight * nChannelNum elements and that the array element type matches ePixelType. *)
		ipImage	:	REFERENCE TO ITcVnImage;	(* Returns the created image (Non-zero interface pointers are reused.) *)
		nWidth	:	UDINT;	(* Image width *)
		nHeight	:	UDINT;	(* Image height *)
		ePixelType	:	ETcVnElementType;	(* Pixel type *)
		nChannelNum	:	UDINT;	(* Number of channels (1 to 255) *)
		hrPrev	:	HRESULT;	(* HRESULT indicating the result of previous operations (If SUCCEEDED(hrPrev) equals false, no operation is executed.) *)
	END_VAR

END_FUNCTION

// Functions/Basic Image Operations/F_VN_ExportImage

	{attribute 'TcIecLibraryType'}
	{attribute 'external_name' := 'F_VN_ExportImage_GUID_CE5F59AA_0180_4944_7A74_96BBB782E30A'}
	(* Exports the image data into a given buffer (e.g. an array). F_VN_ExportImageSize should be called before to get the required buffer size. *)
	FUNCTION F_VN_ExportImage : HRESULT
	VAR_INPUT
		ipImage	:	ITcVnImage;	(* Image *)
		pBuffer	:	PVOID;	(* Pointer to a buffer to store the image data (Make sure to allocate enough memory! The required size in bytes can be determined using the function F_VN_ExportImageSize) *)
		nBufferSize	:	ULINT;	(* Size of the buffer memory in bytes *)
		hrPrev	:	HRESULT;	(* HRESULT indicating the result of previous operations (If SUCCEEDED(hrPrev) equals false, no operation is executed.) *)
	END_VAR

END_FUNCTION

// Functions/Basic Image Operations/F_VN_ExportImageSize

	{attribute 'TcIecLibraryType'}
	{attribute 'external_name' := 'F_VN_ExportImageSize_GUID_45E0275C_F357_4607_5D16_50D5DCBEBC49'}
	(* Get the required buffer size (in bytes) to store the image data. *)
	FUNCTION F_VN_ExportImageSize : HRESULT
	VAR_INPUT
		ipImage	:	ITcVnImage;	(* Image *)
		nBufferSize	:	REFERENCE TO ULINT;	(* Returns the required buffer size in bytes *)
		hrPrev	:	HRESULT;	(* HRESULT indicating the result of previous operations (If SUCCEEDED(hrPrev) equals false, no operation is executed.) *)
	END_VAR

END_FUNCTION

// Functions/Basic Image Operations/F_VN_ExportImageAsBmp

	{attribute 'TcIecLibraryType'}
	{attribute 'external_name' := 'F_VN_ExportImageAsBmp_GUID_9706AE85_D514_47FE_54B3_2856A32D7072'}
	(* Exports the image as bitmap into a given buffer (e.g. an array). F_VN_ExportImageAsBmpSize should be called before to get the required buffer size. *)
	FUNCTION F_VN_ExportImageAsBmp : HRESULT
	VAR_INPUT
		ipImage	:	ITcVnImage;	(* Image *)
		pBuffer	:	PVOID;	(* Pointer to a buffer to store the bitmap image (Make sure to allocate enough memory! The required size in bytes can be determined using the function F_VN_ExportImageAsBmpSize) *)
		nBufferSize	:	ULINT;	(* Size of the buffer memory in bytes *)
		hrPrev	:	HRESULT;	(* HRESULT indicating the result of previous operations (If SUCCEEDED(hrPrev) equals false, no operation is executed.) *)
	END_VAR

END_FUNCTION

// Functions/Basic Image Operations/F_VN_ExportImageAsBmpSize

	{attribute 'TcIecLibraryType'}
	{attribute 'external_name' := 'F_VN_ExportImageAsBmpSize_GUID_D315D7BC_DBFE_4A93_4E8A_9340E24A4D3E'}
	(* Get the required buffer size (in bytes) to store the image as bitmap. *)
	FUNCTION F_VN_ExportImageAsBmpSize : HRESULT
	VAR_INPUT
		ipImage	:	ITcVnImage;	(* Image *)
		nBufferSize	:	REFERENCE TO ULINT;	(* Returns the required buffer size in bytes *)
		hrPrev	:	HRESULT;	(* HRESULT indicating the result of previous operations (If SUCCEEDED(hrPrev) equals false, no operation is executed.) *)
	END_VAR

END_FUNCTION

// Functions/Basic Image Operations/F_VN_ExportImageAsBmpExp

	{attribute 'TcIecLibraryType'}
	{attribute 'external_name' := 'F_VN_ExportImageAsBmpExp_GUID_9BBF3AB7_D620_4EA3_6769_4BED56DED7E4'}
	(* Exports the image as bitmap into a given buffer (e.g. an array). F_VN_ExportImageAsBmpSizeExp should be called before to get the required buffer size. (expert function) *)
	FUNCTION F_VN_ExportImageAsBmpExp : HRESULT
	VAR_INPUT
		ipImage	:	ITcVnImage;	(* Image *)
		pBuffer	:	PVOID;	(* Pointer to a buffer to store the bitmap image (Make sure to allocate enough memory! The required size in bytes can be determined using the function F_VN_ExportImageAsBmpSizeExp) *)
		nBufferSize	:	ULINT;	(* Size of the buffer memory in bytes *)
		nWidth	:	UDINT;	(* Desired width (or 0 to keep the original width) *)
		nHeight	:	UDINT;	(* Desired height (or 0 to keep the original height) *)
		hrPrev	:	HRESULT;	(* HRESULT indicating the result of previous operations (If SUCCEEDED(hrPrev) equals false, no operation is executed.) *)
	END_VAR

END_FUNCTION

// Functions/Basic Image Operations/F_VN_ExportImageAsBmpSizeExp

	{attribute 'TcIecLibraryType'}
	{attribute 'external_name' := 'F_VN_ExportImageAsBmpSizeExp_GUID_C9E6A772_15E9_4C36_5B73_488D17ADEF1A'}
	(* Get the required buffer size (in bytes) to store the image as bitmap. (expert function) *)
	FUNCTION F_VN_ExportImageAsBmpSizeExp : HRESULT
	VAR_INPUT
		ipImage	:	ITcVnImage;	(* Image *)
		nBufferSize	:	REFERENCE TO ULINT;	(* Returns the required buffer size in bytes *)
		nWidth	:	UDINT;	(* Desired width (or 0 to keep the original width) *)
		nHeight	:	UDINT;	(* Desired height (or 0 to keep the original height) *)
		hrPrev	:	HRESULT;	(* HRESULT indicating the result of previous operations (If SUCCEEDED(hrPrev) equals false, no operation is executed.) *)
	END_VAR

END_FUNCTION

// Functions/Basic Image Operations/F_VN_FuseImages

	{attribute 'TcIecLibraryType'}
	{attribute 'external_name' := 'F_VN_FuseImages_GUID_983B1192_98DF_491B_45F6_0765041EAE78'}
	(* Fuse 2 images vertically (intended for line scan cameras). *)
	FUNCTION F_VN_FuseImages : HRESULT
	VAR_INPUT
		ipSrcImage1	:	ITcVnImage;	(* Source image 1 *)
		ipSrcImage2	:	ITcVnImage;	(* Source image 2 *)
		ipDestImage	:	REFERENCE TO ITcVnImage;	(* Destination image *)
		nFirstLine	:	UDINT;	(* Line index in ipSrcImage1, which is the first line in ipDestImage *)
		nNumLines	:	UDINT;	(* The number of lines that should be copied to ipDestImage, starting with nFirstLine in ipSrcImage1. Once the last line of ipSrcImage1 was copied, the remaining lines are copied from ipSrcImage2, starting at line index 0. *)
		hrPrev	:	HRESULT;	(* HRESULT indicating the result of previous operations (If SUCCEEDED(hrPrev) equals false, no operation is executed.) *)
	END_VAR

END_FUNCTION

// Functions/Basic Image Operations/F_VN_FuseImagesArray

	{attribute 'TcIecLibraryType'}
	{attribute 'external_name' := 'F_VN_FuseImagesArray_GUID_AC327679_804E_4E16_411D_08513D7F7B32'}
	(* Fuse up to 10 images vertically (intended for line scan cameras). *)
	FUNCTION F_VN_FuseImagesArray : HRESULT
	VAR_INPUT
		aSrcImageArray	:	REFERENCE TO TcVnArray10_ITcVnImage;	(* Ten-element source image array (not all elements need to be filled, nValidImages specifies the actual amount of images) *)
		nValidImages	:	UDINT;	(* Number of valid images in aSrcImageArray *)
		ipDestImage	:	REFERENCE TO ITcVnImage;	(* Destination image *)
		nFirstLine	:	UDINT;	(* Line index in ipSrcImage1, which is the first line in ipDestImage *)
		nNumLines	:	UDINT;	(* The number of lines that should be copied to ipDestImage, starting with nFirstLine in aSrcImageArray[0]. Once the last line of aSrcImageArray[0] was copied, the remaining lines are copied from aSrcImageArray[1] (starting at line index 0) and so on. *)
		hrPrev	:	HRESULT;	(* HRESULT indicating the result of previous operations (If SUCCEEDED(hrPrev) equals false, no operation is executed.) *)
	END_VAR

END_FUNCTION

// Functions/Basic Image Operations/F_VN_GetImageChannel

	{attribute 'TcIecLibraryType'}
	{attribute 'external_name' := 'F_VN_GetImageChannel_GUID_C9D50485_B845_4A90_7C8A_B2479D97C3C1'}
	(* Return the specified source image channel as a single-channel image. *)
	FUNCTION F_VN_GetImageChannel : HRESULT
	VAR_INPUT
		ipSrcImage	:	ITcVnImage;	(* Source image *)
		ipDestImage	:	REFERENCE TO ITcVnImage;	(* Destination image (An appropriate image will be created if required.) *)
		nChannelIndex	:	UINT;	(* Index of the requested source image channel *)
		hrPrev	:	HRESULT;	(* HRESULT indicating the result of previous operations (If SUCCEEDED(hrPrev) equals false, no operation is executed.) *)
	END_VAR

END_FUNCTION

// Functions/Basic Image Operations/F_VN_GetImageHeight

	{attribute 'TcIecLibraryType'}
	{attribute 'external_name' := 'F_VN_GetImageHeight_GUID_B913C4C4_BF6F_49F8_72C9_726B1145BA99'}
	(* Return the height of an image. (Alternatively use interface method .GetHeight.) *)
	FUNCTION F_VN_GetImageHeight : HRESULT
	VAR_INPUT
		ipImage	:	ITcVnImage;	(* Image *)
		nHeight	:	REFERENCE TO UDINT;	(* Return the height of ipImage *)
		hrPrev	:	HRESULT;	(* HRESULT indicating the result of previous operations (If SUCCEEDED(hrPrev) equals false, no operation is executed.) *)
	END_VAR

END_FUNCTION

// Functions/Basic Image Operations/F_VN_GetImageInfo

	{attribute 'TcIecLibraryType'}
	{attribute 'external_name' := 'F_VN_GetImageInfo_GUID_F85E4AD2_FB0B_4E74_6327_4822A73B67EA'}
	(* Gets a struct containing all common meta infos of the image. (Alternatively use interface method .GetImageInfo.) *)
	FUNCTION F_VN_GetImageInfo : HRESULT
	VAR_INPUT
		ipImage	:	ITcVnImage;	(* Image *)
		stImageInfo	:	REFERENCE TO TcVnImageInfo;	(* Returns a struct describing the image *)
		hrPrev	:	HRESULT;	(* HRESULT indicating the result of previous operations (If SUCCEEDED(hrPrev) equals false, no operation is executed.) *)
	END_VAR

END_FUNCTION

// Functions/Basic Image Operations/F_VN_GetImageWidth

	{attribute 'TcIecLibraryType'}
	{attribute 'external_name' := 'F_VN_GetImageWidth_GUID_81F138A3_8A5D_45FE_6E1D_E90491D52173'}
	(* Return the width of an image. (Alternatively use interface method .GetWidth.) *)
	FUNCTION F_VN_GetImageWidth : HRESULT
	VAR_INPUT
		ipImage	:	ITcVnImage;	(* Image *)
		nWidth	:	REFERENCE TO UDINT;	(* Return the width of ipImage *)
		hrPrev	:	HRESULT;	(* HRESULT indicating the result of previous operations (If SUCCEEDED(hrPrev) equals false, no operation is executed.) *)
	END_VAR

END_FUNCTION

// Functions/Basic Image Operations/F_VN_GetPixel

	{attribute 'TcIecLibraryType'}
	{attribute 'external_name' := 'F_VN_GetPixel_GUID_8318349B_840C_4F9E_7944_52E9B6DD3156'}
	(* Gets a specific pixel. *)
	FUNCTION F_VN_GetPixel : HRESULT
	VAR_INPUT
		ipSrcImage	:	ITcVnImage;	(* Source image *)
		aValue	:	REFERENCE TO TcVnVector4_LREAL;	(* Returns the pixel value (Unused channels are set to 0.) *)
		nX	:	UDINT;	(* x coordinate of the pixel *)
		nY	:	UDINT;	(* y coordinate of the pixel *)
		hrPrev	:	HRESULT;	(* HRESULT indicating the result of previous operations (If SUCCEEDED(hrPrev) equals false, no operation is executed.) *)
	END_VAR

END_FUNCTION

// Functions/Basic Image Operations/F_VN_GetPixelFormat

	{attribute 'TcIecLibraryType'}
	{attribute 'external_name' := 'F_VN_GetPixelFormat_GUID_0810316D_A879_4876_414C_B8E06B9017D5'}
	(* Gets the pixel format of an image. (Alternatively use interface method .GetPixelFormat.) *)
	FUNCTION F_VN_GetPixelFormat : HRESULT
	VAR_INPUT
		ipImage	:	ITcVnImage;	(* Image *)
		stPixelFormat	:	REFERENCE TO TcVnPixelFormat;	(* Returns a struct describing the pixel format *)
		hrPrev	:	HRESULT;	(* HRESULT indicating the result of previous operations (If SUCCEEDED(hrPrev) equals false, no operation is executed.) *)
	END_VAR

END_FUNCTION

// Functions/Basic Image Operations/F_VN_GetRoi

	{attribute 'TcIecLibraryType'}
	{attribute 'external_name' := 'F_VN_GetRoi_GUID_CBB4A4C8_02EC_4C71_7A36_30B16F8ACA9F'}
	(* Gets the coordinates of the region of interest (ROI) within the image. *)
	FUNCTION F_VN_GetRoi : HRESULT
	VAR_INPUT
		ipSrcImage	:	ITcVnImage;	(* Source image *)
		stRoi	:	REFERENCE TO TcVnRectangle_UDINT;	(* Returns the coordinates of the region of interest *)
		hrPrev	:	HRESULT;	(* HRESULT indicating the result of previous operations (If SUCCEEDED(hrPrev) equals false, no operation is executed.) *)
	END_VAR

END_FUNCTION

// Functions/Basic Image Operations/F_VN_MixImageChannels

	{attribute 'TcIecLibraryType'}
	{attribute 'external_name' := 'F_VN_MixImageChannels_GUID_CD34034C_3D11_4661_5829_BD624E44D8AD'}
	(* Mix image channels by copying the specified channels of the source image into the specified channels of the destination image. *)
	FUNCTION F_VN_MixImageChannels : HRESULT
	VAR_INPUT
		ipSrcImage	:	ITcVnImage;	(* Source image *)
		ipDestImage	:	REFERENCE TO ITcVnImage;	(* Destination image (An appropriate image will be created if required.) *)
		ipIndicesFromTo	:	ITcVnContainer;	(* Index pairs (ContainerType_Vector_TcVnVector2_DINT), specifying which source channel (TcVnVector2_DINT [0]) should be copied to which destination channel (TcVnVector2_DINT [1]). *)
		hrPrev	:	HRESULT;	(* HRESULT indicating the result of previous operations (If SUCCEEDED(hrPrev) equals false, no operation is executed.) *)
	END_VAR

END_FUNCTION

// Functions/Basic Image Operations/F_VN_ResetRoi

	{attribute 'TcIecLibraryType'}
	{attribute 'external_name' := 'F_VN_ResetRoi_GUID_1B2497BF_253A_42A2_67C6_7CB9E6A3279C'}
	(* Reset the region of interest (ROI) of an image. (After this operation, the ROI is set to the entire image.) *)
	FUNCTION F_VN_ResetRoi : HRESULT
	VAR_INPUT
		ipImage	:	ITcVnImage;	(* Image *)
		hrPrev	:	HRESULT;	(* HRESULT indicating the result of previous operations (If SUCCEEDED(hrPrev) equals false, no operation is executed.) *)
	END_VAR

END_FUNCTION

// Functions/Basic Image Operations/F_VN_SetImageChannel

	{attribute 'TcIecLibraryType'}
	{attribute 'external_name' := 'F_VN_SetImageChannel_GUID_3D65BE46_78B1_4B82_4FB7_45F04ADAE799'}
	(* Sets the specified destination image channel to the values of the specified source image channel. *)
	FUNCTION F_VN_SetImageChannel : HRESULT
	VAR_INPUT
		ipSrcImage	:	ITcVnImage;	(* Source image *)
		ipDestImage	:	REFERENCE TO ITcVnImage;	(* Destination image (An appropriate image will be created if required.) *)
		nSrcChannelIndex	:	UINT;	(* Index of the source image channel *)
		nDestChannelIndex	:	UINT;	(* Index of the destination image channel, which will be replaced by the specified source image channel *)
		hrPrev	:	HRESULT;	(* HRESULT indicating the result of previous operations (If SUCCEEDED(hrPrev) equals false, no operation is executed.) *)
	END_VAR

END_FUNCTION

// Functions/Basic Image Operations/F_VN_SetPixel

	{attribute 'TcIecLibraryType'}
	{attribute 'external_name' := 'F_VN_SetPixel_GUID_BC30965F_22FD_4FD8_68B1_EEB11291FEAA'}
	(* Sets a specific pixel. *)
	FUNCTION F_VN_SetPixel : HRESULT
	VAR_INPUT
		ipSrcImage	:	ITcVnImage;	(* Source image *)
		aValue	:	REFERENCE TO TcVnVector4_LREAL;	(* The pixel value to set (additional channels are ignored.) *)
		nX	:	UDINT;	(* x coordinate of the pixel *)
		nY	:	UDINT;	(* y coordinate of the pixel *)
		hrPrev	:	HRESULT;	(* HRESULT indicating the result of previous operations (If SUCCEEDED(hrPrev) equals false, no operation is executed.) *)
	END_VAR

END_FUNCTION

// Functions/Basic Image Operations/F_VN_SetPixels

	{attribute 'TcIecLibraryType'}
	{attribute 'external_name' := 'F_VN_SetPixels_GUID_CD97B4BB_462C_411C_6E5A_F4EF3392D595'}
	(* Sets all pixels of an image to a given value. *)
	FUNCTION F_VN_SetPixels : HRESULT
	VAR_INPUT
		ipDestImage	:	ITcVnImage;	(* Destination image *)
		aValue	:	REFERENCE TO TcVnVector4_LREAL;	(* Pixel value *)
		hrPrev	:	HRESULT;	(* HRESULT indicating the result of previous operations (If SUCCEEDED(hrPrev) equals false, no operation is executed.) *)
	END_VAR

END_FUNCTION

// Functions/Basic Image Operations/F_VN_SetPixelsExp

	{attribute 'TcIecLibraryType'}
	{attribute 'external_name' := 'F_VN_SetPixelsExp_GUID_72BFAAF4_6001_4DB0_7AC3_01F7F510700F'}
	(* Sets all pixels of an image to a given value. (expert function) *)
	FUNCTION F_VN_SetPixelsExp : HRESULT
	VAR_INPUT
		ipDestImage	:	ITcVnImage;	(* Destination image *)
		aValue	:	REFERENCE TO TcVnVector4_LREAL;	(* Pixel value *)
		ipMask	:	ITcVnImage;	(* Mask image *)
		hrPrev	:	HRESULT;	(* HRESULT indicating the result of previous operations (If SUCCEEDED(hrPrev) equals false, no operation is executed.) *)
	END_VAR

END_FUNCTION

// Functions/Basic Image Operations/F_VN_SetRoi

	{attribute 'TcIecLibraryType'}
	{attribute 'external_name' := 'F_VN_SetRoi_GUID_5C2B00B1_F0D3_4BC3_725E_C72AC2888DAF'}
	(* Sets a region of interest (ROI) within an image. *)
	FUNCTION F_VN_SetRoi : HRESULT
	VAR_INPUT
		nX	:	UDINT;	(* Left boundary (inclusive 0-based index) *)
		nY	:	UDINT;	(* Upper boundary (inclusive 0-based index) *)
		nWidth	:	UDINT;	(* ROI width *)
		nHeight	:	UDINT;	(* ROI height *)
		ipDestImage	:	ITcVnImage;	(* Destination image *)
		hrPrev	:	HRESULT;	(* HRESULT indicating the result of previous operations (If SUCCEEDED(hrPrev) equals false, no operation is executed.) *)
	END_VAR

END_FUNCTION

// Functions/Basic Image Operations/F_VN_SetRoi_TcVnRectangle_UDINT

